C01808=1056.490,410.980,-122.148,174.990,39.875,157.709
C01809=1056.498,411.227,-122.192,174.998,39.884,157.712
C01810=1056.506,411.473,-122.237,175.006,39.892,157.714
C01811=1056.516,411.718,-122.281,175.013,39.901,157.717
C01812=1056.525,411.964,-122.327,175.022,39.910,157.719
C01813=1056.534,412.210,-122.372,175.029,39.918,157.722
C01814=1056.543,412.455,-122.416,175.037,39.927,157.724
C01815=1056.552,412.702,-122.461,175.045,39.935,157.727
C01816=1056.561,412.947,-122.506,175.053,39.944,157.730
C01817=1056.570,413.193,-122.552,175.062,39.953,157.732
C01818=1056.579,413.439,-122.596,175.069,39.962,157.735
C01819=1056.588,413.685,-122.641,175.077,39.970,157.737
C01820=1056.596,413.930,-122.686,175.086,39.980,157.740
C01821=1056.605,414.176,-122.732,175.093,39.989,157.743
C01822=1056.614,414.422,-122.777,175.102,39.997,157.745
C01823=1056.623,414.668,-122.822,175.110,40.007,157.748
C01824=1056.632,414.914,-122.868,175.118,40.015,157.750
C01825=1056.641,415.159,-122.913,175.126,40.025,157.753
C01826=1056.650,415.405,-122.959,175.135,40.033,157.756
C01827=1056.659,415.650,-123.004,175.143,40.043,157.758
C01828=1056.668,415.896,-123.050,175.151,40.052,157.761
C01829=1056.680,416.243,-123.114,175.163,40.065,157.765
C01830=1056.694,416.590,-123.179,175.174,40.078,157.769
C01831=1056.706,416.937,-123.244,175.186,40.090,157.772
C01832=1056.719,417.283,-123.308,175.198,40.103,157.776
C01833=1056.728,417.529,-123.354,175.207,40.112,157.779
C01834=1056.737,417.774,-123.400,175.216,40.122,157.782
C01835=1056.746,418.020,-123.445,175.224,40.131,157.785
C01836=1056.756,418.265,-123.491,175.233,40.141,157.787
C01837=1056.765,418.512,-123.537,175.241,40.150,157.790
C01838=1056.774,418.757,-123.583,175.249,40.159,157.793
C01839=1056.783,419.002,-123.630,175.258,40.169,157.796
C01840=1056.792,419.248,-123.675,175.267,40.178,157.798
C01841=1056.801,419.493,-123.722,175.276,40.188,157.801
C01842=1056.811,419.739,-123.768,175.284,40.197,157.804
C01843=1056.820,419.985,-123.814,175.293,40.207,157.807
C01844=1056.830,420.230,-123.860,175.302,40.216,157.810
C01845=1056.839,420.476,-123.907,175.311,40.225,157.813
C01846=1056.848,420.721,-123.954,175.319,40.235,157.815
C01847=1056.857,420.967,-124.000,175.328,40.245,157.818
C01848=1056.866,421.212,-124.046,175.337,40.254,157.821
C01849=1056.876,421.458,-124.093,175.346,40.264,157.824
C01850=1056.884,421.703,-124.140,175.355,40.274,157.827
C01851=1056.894,421.949,-124.186,175.364,40.283,157.830
C01852=1056.904,422.194,-124.233,175.373,40.293,157.833
C01853=1056.912,422.439,-124.280,175.383,40.303,157.836
C01854=1056.922,422.685,-124.326,175.392,40.313,157.839
C01855=1056.932,422.930,-124.373,175.401,40.323,157.842
C01856=1056.941,423.176,-124.420,175.409,40.333,157.845
C01857=1056.950,423.421,-124.466,175.418,40.343,157.848
C01858=1056.960,423.667,-124.514,175.427,40.353,157.851
C01859=1056.969,423.912,-124.560,175.437,40.363,157.854
C01860=1056.979,424.157,-124.607,175.447,40.372,157.857
C01861=1056.988,424.402,-124.655,175.456,40.382,157.860
C01862=1056.998,424.648,-124.701,175.465,40.393,157.863
C01863=1057.007,424.894,-124.749,175.474,40.403,157.866
C01864=1057.017,425.138,-124.796,175.484,40.413,157.869
C01865=1057.026,425.384,-124.843,175.493,40.423,157.872
C01866=1057.036,425.630,-124.890,175.502,40.433,157.875
C01867=1057.046,425.875,-124.938,175.512,40.443,157.878
C01868=1057.055,426.120,-124.985,175.521,40.453,157.882
C01869=1057.065,426.366,-125.033,175.531,40.463,157.885
C01870=1057.075,426.611,-125.080,175.541,40.474,157.888
C01871=1057.084,426.856,-125.128,175.550,40.484,157.891
C01872=1057.093,427.101,-125.175,175.560,40.495,157.894
C01873=1057.104,427.347,-125.223,175.570,40.505,157.897
C01874=1057.113,427.592,-125.270,175.579,40.515,157.901
C01875=1057.123,427.837,-125.319,175.589,40.526,157.904
C01876=1057.133,428.082,-125.366,175.598,40.537,157.907
C01877=1057.142,428.327,-125.414,175.609,40.547,157.910
C01878=1057.152,428.572,-125.462,175.618,40.558,157.914
C01879=1057.162,428.818,-125.509,175.628,40.568,157.917
C01880=1057.171,429.063,-125.558,175.638,40.579,157.920
C01881=1057.181,429.308,-125.606,175.648,40.590,157.923
C01882=1057.191,429.553,-125.654,175.659,40.600,157.927
C01883=1057.201,429.798,-125.701,175.668,40.611,157.930
C01884=1057.211,430.043,-125.750,175.678,40.622,157.933
C01885=1057.226,430.412,-125.822,175.693,40.638,157.938
C01886=1057.241,430.780,-125.896,175.709,40.654,157.943
C01887=1057.255,431.149,-125.968,175.724,40.670,157.948
C01888=1057.270,431.517,-126.041,175.739,40.687,157.954
C01889=1057.280,431.762,-126.089,175.750,40.698,157.957
C01890=1057.290,432.007,-126.138,175.760,40.709,157.960
C01891=1057.300,432.251,-126.186,175.770,40.720,157.964
C01892=1057.310,432.497,-126.235,175.781,40.731,157.967
C01893=1057.320,432.742,-126.284,175.791,40.742,157.971
C01894=1057.330,432.987,-126.332,175.802,40.753,157.974
C01895=1057.340,433.231,-126.381,175.813,40.765,157.978
C01896=1057.350,433.477,-126.430,175.822,40.776,157.981
C01897=1057.360,433.722,-126.479,175.833,40.787,157.985
C01898=1057.370,433.966,-126.528,175.844,40.798,157.988
C01899=1057.380,434.212,-126.577,175.855,40.810,157.992
C01900=1057.390,434.456,-126.626,175.865,40.821,157.996
C01901=1057.401,434.702,-126.675,175.876,40.833,157.999
C01902=1057.411,434.947,-126.724,175.887,40.843,158.003
C01903=1057.421,435.191,-126.774,175.898,40.855,158.006
C01904=1057.431,435.437,-126.823,175.909,40.867,158.010
C01905=1057.441,435.681,-126.872,175.920,40.878,158.014
C01906=1057.452,435.926,-126.921,175.931,40.890,158.017
C01907=1057.462,436.171,-126.971,175.942,40.901,158.021
C01908=1057.473,436.415,-127.020,175.952,40.913,158.025
C01909=1057.483,436.660,-127.070,175.964,40.924,158.028
C01910=1057.494,436.905,-127.119,175.975,40.936,158.032
C01911=1057.504,437.150,-127.169,175.986,40.948,158.036
C01912=1057.515,437.395,-127.218,175.998,40.959,158.040
C01913=1057.525,437.640,-127.269,176.009,40.971,158.043
C01914=1057.535,437.885,-127.318,176.021,40.983,158.047
C01915=1057.545,438.130,-127.367,176.032,40.995,158.051
C01916=1057.556,438.374,-127.418,176.043,41.007,158.055
C01917=1057.566,438.619,-127.468,176.055,41.019,158.059
C01918=1057.577,438.863,-127.518,176.066,41.031,158.063
C01919=1057.587,439.108,-127.567,176.077,41.043,158.066
C01920=1057.598,439.353,-127.618,176.089,41.055,158.070
C01921=1057.608,439.598,-127.668,176.101,41.067,158.074
C01922=1057.619,439.842,-127.718,176.112,41.079,158.078
C01923=1057.630,440.087,-127.769,176.124,41.092,158.082
C01924=1057.640,440.332,-127.820,176.135,41.104,158.086
C01925=1057.650,440.576,-127.869,176.148,41.116,158.090
C01926=1057.661,440.820,-127.919,176.159,41.128,158.094
C01927=1057.672,441.065,-127.970,176.171,41.141,158.098
C01928=1057.683,441.310,-128.020,176.183,41.153,158.102
C01929=1057.693,441.554,-128.071,176.195,41.166,158.106
C01930=1057.704,441.799,-128.122,176.208,41.178,158.110
C01931=1057.715,442.044,-128.172,176.219,41.190,158.114
C01932=1057.726,442.288,-128.224,176.232,41.203,158.118
C01933=1057.737,442.532,-128.274,176.244,41.216,158.123
C01934=1057.747,442.777,-128.325,176.257,41.228,158.127
C01935=1057.758,443.021,-128.376,176.268,41.241,158.131
C01936=1057.769,443.266,-128.428,176.281,41.254,158.135
C01937=1057.780,443.511,-128.478,176.293,41.266,158.139
C01938=1057.791,443.755,-128.529,176.306,41.279,158.143
C01939=1057.802,443.999,-128.580,176.318,41.292,158.148
C01940=1057.813,444.244,-128.632,176.330,41.305,158.152
C01941=1057.823,444.475,-128.680,176.343,41.317,158.156
C01942=1057.834,444.706,-128.729,176.355,41.329,158.160
C01943=1057.844,444.938,-128.778,176.366,41.341,158.164
C01944=1057.854,445.168,-128.826,176.378,41.354,158.168
C01945=1057.865,445.400,-128.875,176.391,41.366,158.172
C01946=1057.875,445.631,-128.924,176.403,41.378,158.176
C01947=1057.886,445.863,-128.973,176.415,41.391,158.181
C01948=1057.897,446.094,-129.022,176.427,41.404,158.185
C01949=1057.908,446.338,-129.073,176.440,41.417,158.189
C01950=1057.919,446.581,-129.125,176.453,41.430,158.193
C01951=1057.930,446.825,-129.176,176.467,41.443,158.198
C01952=1057.942,447.070,-129.228,176.480,41.456,158.202
C01953=1057.954,447.313,-129.279,176.493,41.469,158.207
C01954=1057.968,447.556,-129.329,176.506,41.482,158.211
C01955=1057.982,447.800,-129.379,176.520,41.495,158.215
C01956=1057.996,448.045,-129.428,176.533,41.507,158.220
C01957=1058.013,448.300,-129.478,176.547,41.519,158.224
C01958=1058.030,448.556,-129.529,176.562,41.532,158.228
C01959=1058.049,448.812,-129.577,176.576,41.544,158.233
C01960=1058.068,449.068,-129.626,176.590,41.556,158.237
C01961=1058.087,449.313,-129.673,176.604,41.568,158.241
C01962=1058.108,449.558,-129.718,176.618,41.578,158.245
C01963=1058.129,449.804,-129.763,176.632,41.589,158.249
C01964=1058.151,450.049,-129.807,176.646,41.600,158.252
C01965=1057.824,450.063,-130.090,176.642,41.708,158.282
C01966=1057.802,449.819,-130.046,176.628,41.698,158.279
C01967=1057.781,449.573,-130.001,176.614,41.687,158.275
C01968=1057.760,449.328,-129.956,176.600,41.676,158.271
C01969=1057.741,449.083,-129.911,176.586,41.665,158.267
C01970=1057.722,448.838,-129.864,176.572,41.653,158.263
C01971=1057.704,448.593,-129.816,176.558,41.641,158.259
C01972=1057.687,448.349,-129.769,176.545,41.630,158.255
C01973=1057.671,448.104,-129.720,176.531,41.618,158.250
C01974=1057.656,447.860,-129.672,176.517,41.606,158.246
C01975=1057.641,447.616,-129.622,176.504,41.593,158.242
C01976=1057.627,447.372,-129.572,176.491,41.581,158.238
C01977=1057.614,447.129,-129.522,176.477,41.568,158.233
C01978=1057.603,446.885,-129.470,176.464,41.555,158.229
C01979=1057.592,446.641,-129.418,176.450,41.542,158.224
C01980=1057.580,446.398,-129.367,176.437,41.528,158.220
C01981=1057.569,446.154,-129.315,176.424,41.515,158.216
C01982=1057.558,445.927,-129.267,176.412,41.503,158.211
C01983=1057.548,445.700,-129.220,176.400,41.491,158.207
C01984=1057.538,445.472,-129.171,176.388,41.479,158.203
C01985=1057.527,445.244,-129.123,176.376,41.467,158.199
C01986=1057.517,445.018,-129.076,176.364,41.455,158.195
C01987=1057.507,444.790,-129.027,176.353,41.442,158.191
C01988=1057.497,444.563,-128.980,176.340,41.430,158.187
C01989=1057.486,444.335,-128.932,176.328,41.419,158.183
C01990=1057.475,444.091,-128.880,176.315,41.406,158.179
C01991=1057.465,443.846,-128.829,176.303,41.393,158.175
C01992=1057.453,443.602,-128.778,176.291,41.380,158.171
C01993=1057.443,443.358,-128.726,176.279,41.368,158.166
C01994=1057.432,443.113,-128.676,176.266,41.355,158.162
C01995=1057.421,442.869,-128.624,176.253,41.342,158.158
C01996=1057.410,442.624,-128.574,176.241,41.330,158.154
C01997=1057.399,442.379,-128.523,176.229,41.317,158.150
C01998=1057.382,441.999,-128.444,176.210,41.298,158.143
C01999=1057.365,441.618,-128.364,176.191,41.278,158.137
C02000=1057.348,441.236,-128.286,176.172,41.259,158.131
C02001=1057.332,440.856,-128.207,176.154,41.240,158.124
C02002=1057.321,440.611,-128.156,176.141,41.228,158.120
C02003=1057.310,440.367,-128.105,176.129,41.216,158.116
C02004=1057.299,440.122,-128.055,176.118,41.203,158.112
C02005=1057.289,439.877,-128.005,176.105,41.191,158.108
C02006=1057.279,439.633,-127.955,176.094,41.179,158.104
C02007=1057.268,439.389,-127.905,176.082,41.167,158.100
C02008=1057.257,439.144,-127.855,176.071,41.155,158.096
C02009=1057.247,438.899,-127.804,176.059,41.143,158.093
C02010=1057.237,438.654,-127.754,176.047,41.131,158.089
C02011=1057.226,438.409,-127.704,176.036,41.119,158.085
C02012=1057.215,438.164,-127.655,176.024,41.107,158.081
C02013=1057.205,437.920,-127.604,176.013,41.096,158.077
C02014=1057.195,437.675,-127.554,176.002,41.084,158.074
C02015=1057.184,437.430,-127.505,175.991,41.072,158.070
C02016=1057.174,437.186,-127.456,175.979,41.060,158.066
C02017=1057.163,436.941,-127.406,175.968,41.048,158.062
C02018=1057.152,436.696,-127.356,175.957,41.037,158.058
C02019=1057.142,436.451,-127.306,175.946,41.025,158.055
C02020=1057.132,436.206,-127.257,175.934,41.014,158.051
C02021=1057.121,435.961,-127.208,175.923,41.002,158.047
C02022=1057.111,435.717,-127.159,175.912,40.991,158.044
C02023=1057.100,435.472,-127.109,175.901,40.979,158.040
C02024=1057.090,435.227,-127.060,175.890,40.967,158.036
C02025=1057.080,434.982,-127.010,175.879,40.956,158.033
C02026=1057.070,434.737,-126.962,175.868,40.945,158.029
C02027=1057.059,434.492,-126.912,175.857,40.934,158.025
C02028=1057.049,434.247,-126.863,175.847,40.922,158.022
C02029=1057.039,434.002,-126.814,175.836,40.911,158.018
C02030=1057.029,433.758,-126.765,175.825,40.900,158.015
C02031=1057.019,433.513,-126.716,175.814,40.889,158.011
C02032=1057.009,433.267,-126.667,175.804,40.877,158.008
C02033=1056.999,433.023,-126.618,175.793,40.866,158.004
C02034=1056.989,432.778,-126.569,175.782,40.855,158.001
C02035=1056.978,432.532,-126.521,175.771,40.844,157.997
C02036=1056.969,432.287,-126.472,175.762,40.833,157.994
C02037=1056.959,432.043,-126.423,175.751,40.822,157.990
C02038=1056.949,431.803,-126.375,175.741,40.811,157.987
C02039=1056.939,431.564,-126.328,175.730,40.801,157.983
C02040=1056.929,431.325,-126.280,175.720,40.790,157.980
C02041=1056.920,431.086,-126.233,175.711,40.779,157.977
C02042=1056.910,430.846,-126.186,175.700,40.769,157.973
C02043=1056.901,430.607,-126.138,175.691,40.758,157.970
C02044=1056.891,430.367,-126.092,175.680,40.748,157.967
C02045=1056.882,430.128,-126.044,175.670,40.737,157.964
C02046=1056.872,429.883,-125.996,175.661,40.726,157.960
C02047=1056.862,429.638,-125.948,175.650,40.716,157.957
C02048=1056.852,429.393,-125.900,175.640,40.705,157.954
C02049=1056.842,429.147,-125.852,175.630,40.695,157.950
C02050=1056.832,428.903,-125.804,175.620,40.684,157.947
C02051=1056.822,428.657,-125.756,175.611,40.673,157.944
C02052=1056.813,428.412,-125.708,175.600,40.663,157.940
C02053=1056.803,428.167,-125.660,175.591,40.652,157.937
C02054=1056.793,427.922,-125.612,175.580,40.642,157.934
C02055=1056.783,427.676,-125.564,175.571,40.632,157.931
C02056=1056.773,427.431,-125.517,175.561,40.621,157.928
C02057=1056.764,427.185,-125.469,175.552,40.611,157.924
C02058=1056.754,426.940,-125.421,175.541,40.601,157.921
C02059=1056.744,426.696,-125.374,175.532,40.590,157.918
C02060=1056.735,426.450,-125.326,175.522,40.580,157.915
C02061=1056.725,426.205,-125.278,175.513,40.570,157.912
C02062=1056.715,425.959,-125.231,175.503,40.559,157.908
C02063=1056.706,425.714,-125.183,175.493,40.549,157.905
C02064=1056.696,425.469,-125.136,175.484,40.539,157.902
C02065=1056.687,425.223,-125.089,175.474,40.529,157.899
C02066=1056.677,424.978,-125.042,175.465,40.519,157.896
C02067=1056.667,424.733,-124.995,175.456,40.509,157.893
C02068=1056.658,424.487,-124.947,175.447,40.499,157.890
C02069=1056.648,424.242,-124.901,175.437,40.489,157.887
C02070=1056.639,423.997,-124.853,175.428,40.479,157.884
C02071=1056.629,423.751,-124.806,175.418,40.469,157.881
C02072=1056.620,423.506,-124.760,175.408,40.459,157.878
C02073=1056.610,423.261,-124.712,175.399,40.449,157.875
C02074=1056.601,423.015,-124.666,175.390,40.439,157.872
C02075=1056.591,422.770,-124.618,175.381,40.430,157.869
C02076=1056.582,422.525,-124.572,175.372,40.420,157.866
C02077=1056.572,422.279,-124.526,175.363,40.410,157.863
C02078=1056.563,422.034,-124.478,175.354,40.400,157.860
C02079=1056.553,421.788,-124.432,175.345,40.390,157.857
C02080=1056.544,421.543,-124.386,175.336,40.381,157.854
C02081=1056.536,421.297,-124.339,175.327,40.371,157.851
C02082=1056.526,421.051,-124.292,175.318,40.361,157.848
C02083=1056.517,420.806,-124.246,175.309,40.352,157.845
C02084=1056.508,420.561,-124.199,175.300,40.342,157.842
C02085=1056.498,420.315,-124.152,175.292,40.333,157.840
C02086=1056.489,420.070,-124.105,175.283,40.323,157.837
C02087=1056.480,419.825,-124.059,175.274,40.314,157.834
C02088=1056.470,419.578,-124.014,175.265,40.304,157.831
C02089=1056.461,419.333,-123.967,175.256,40.295,157.828
C02090=1056.452,419.088,-123.921,175.248,40.285,157.825
C02091=1056.442,418.842,-123.875,175.239,40.276,157.823
C02092=1056.433,418.596,-123.829,175.230,40.267,157.820
C02093=1056.424,418.350,-123.783,175.221,40.257,157.817
C02094=1056.415,418.105,-123.737,175.213,40.248,157.814
C02095=1056.406,417.859,-123.691,175.204,40.239,157.812
C02096=1056.397,417.614,-123.645,175.195,40.230,157.809
C02097=1056.388,417.368,-123.600,175.187,40.221,157.806
C02098=1056.375,417.020,-123.534,175.175,40.207,157.802
C02099=1056.361,416.671,-123.469,175.163,40.194,157.798
C02100=1056.348,416.322,-123.405,175.151,40.182,157.794
C02101=1056.336,415.974,-123.339,175.139,40.169,157.791
C02102=1056.327,415.728,-123.294,175.130,40.160,157.788
C02103=1056.318,415.482,-123.248,175.123,40.150,157.785
C02104=1056.309,415.236,-123.203,175.114,40.142,157.783
C02105=1056.300,414.990,-123.158,175.106,40.132,157.780
C02106=1056.291,414.745,-123.112,175.097,40.124,157.777
C02107=1056.282,414.499,-123.066,175.090,40.114,157.775
C02108=1056.273,414.254,-123.021,175.081,40.106,157.772
C02109=1056.264,414.008,-122.975,175.073,40.097,157.769
C02110=1056.255,413.762,-122.930,175.065,40.088,157.767
C02111=1056.247,413.516,-122.885,175.057,40.079,157.764
C02112=1056.237,413.271,-122.841,175.048,40.070,157.762
C02113=1056.228,413.025,-122.795,175.041,40.062,157.759
C02114=1056.219,412.779,-122.750,175.033,40.053,157.757
C02115=1056.211,412.533,-122.705,175.024,40.044,157.754
C02116=1056.201,412.287,-122.660,175.017,40.036,157.751
C02117=1056.192,412.041,-122.615,175.008,40.027,157.749
C02118=1056.184,411.795,-122.570,175.001,40.019,157.746
C02119=1056.174,411.550,-122.526,174.993,40.010,157.744
C02120=1056.165,411.304,-122.480,174.984,40.001,157.741
C02121=1056.157,411.058,-122.436,174.977,39.993,157.739
C02122=1056.148,410.813,-122.390,174.969,39.984,157.736
C02123=1056.139,410.566,-122.346,174.961,39.976,157.734
C02124=1056.131,410.321,-122.302,174.953,39.967,157.731
C02125=1056.122,410.075,-122.257,174.946,39.959,157.729
C02126=1056.112,409.829,-122.213,174.938,39.950,157.727
C02127=1056.104,409.583,-122.168,174.930,39.942,157.724
C02128=1056.095,409.337,-122.123,174.922,39.933,157.722
C02129=1056.086,409.092,-122.079,174.915,39.925,157.719
C02130=1056.078,408.845,-122.034,174.907,39.917,157.717
C02131=1056.069,408.600,-121.991,174.899,39.908,157.714
C02132=1056.060,408.353,-121.946,174.891,39.900,157.712
C02133=1056.052,408.108,-121.902,174.884,39.892,157.710
C02134=1056.043,407.862,-121.857,174.876,39.883,157.707
C02135=1056.034,407.616,-121.812,174.869,39.875,157.705
C02136=1056.026,407.370,-121.768,174.862,39.867,157.702
C02137=1056.017,407.124,-121.724,174.853,39.859,157.700
C02138=1056.009,406.878,-121.680,174.846,39.850,157.698
C02139=1056.000,406.632,-121.636,174.839,39.842,157.695
C02140=1055.992,406.386,-121.592,174.831,39.834,157.693
C02141=1055.984,406.140,-121.548,174.824,39.826,157.691
C02142=1055.974,405.894,-121.503,174.816,39.818,157.688
C02143=1055.966,405.649,-121.459,174.809,39.810,157.686
C02144=1055.958,405.403,-121.416,174.802,39.801,157.684
C02145=1055.950,405.157,-121.372,174.794,39.793,157.681
C02146=1055.940,404.911,-121.328,174.787,39.786,157.679
C02147=1055.932,404.664,-121.284,174.780,39.777,157.677
C02148=1055.924,404.419,-121.240,174.773,39.769,157.674
C02149=1055.916,404.173,-121.196,174.765,39.762,157.672
C02150=1055.906,403.926,-121.152,174.758,39.754,157.670
C02151=1055.898,403.680,-121.109,174.751,39.745,157.668
C02152=1055.890,403.435,-121.065,174.743,39.738,157.665
C02153=1055.881,403.189,-121.022,174.736,39.730,157.663
C02154=1055.870,402.846,-120.961,174.726,39.719,157.660
C02155=1055.857,402.503,-120.901,174.716,39.708,157.657
C02156=1055.846,402.160,-120.840,174.706,39.697,157.654
C02157=1055.835,401.817,-120.780,174.697,39.686,157.651
C02158=1055.826,401.570,-120.736,174.690,39.679,157.649
C02159=1055.817,401.325,-120.693,174.683,39.671,157.646
C02160=1055.809,401.079,-120.650,174.675,39.663,157.644
C02161=1055.800,400.833,-120.606,174.668,39.656,157.642
C02162=1055.792,400.586,-120.563,174.661,39.648,157.640
C02163=1055.784,400.340,-120.520,174.654,39.640,157.638
C02164=1055.775,400.094,-120.477,174.647,39.633,157.636
C02165=1055.767,399.848,-120.434,174.641,39.626,157.634
C02166=1055.758,399.602,-120.391,174.634,39.618,157.631
C02167=1055.750,399.356,-120.348,174.627,39.611,157.629
C02168=1055.742,399.110,-120.306,174.620,39.603,157.627
C02169=1055.734,398.864,-120.262,174.612,39.595,157.625
C02170=1055.726,398.618,-120.219,174.606,39.588,157.623
C02171=1055.717,398.371,-120.176,174.599,39.581,157.621
C02172=1055.709,398.125,-120.133,174.592,39.573,157.619
C02173=1055.701,397.879,-120.091,174.585,39.565,157.617
C02174=1055.693,397.633,-120.048,174.579,39.558,157.615
C02175=1055.684,397.387,-120.005,174.572,39.551,157.612
C02176=1055.676,397.141,-119.963,174.565,39.543,157.610
C02177=1055.668,396.895,-119.920,174.558,39.536,157.608
C02178=1055.660,396.649,-119.878,174.552,39.529,157.606
C02179=1055.652,396.403,-119.835,174.545,39.521,157.604
C02180=1055.643,396.156,-119.792,174.538,39.514,157.602
C02181=1055.635,395.910,-119.749,174.532,39.507,157.600
C02182=1055.627,395.664,-119.707,174.525,39.500,157.598
C02183=1055.619,395.418,-119.664,174.518,39.492,157.596
C02184=1055.611,395.171,-119.622,174.512,39.485,157.594
C02185=1055.603,394.925,-119.580,174.505,39.478,157.592
C02186=1055.594,394.679,-119.538,174.498,39.471,157.590
C02187=1055.586,394.433,-119.495,174.493,39.464,157.588
C02188=1055.578,394.187,-119.454,174.486,39.456,157.586
C02189=1055.570,393.940,-119.411,174.479,39.450,157.584
C02190=1055.562,393.695,-119.369,174.473,39.442,157.582
C02191=1055.554,393.448,-119.326,174.466,39.435,157.580
C02192=1055.546,393.202,-119.284,174.460,39.428,157.578
C02193=1055.537,392.956,-119.243,174.453,39.421,157.576
C02194=1055.530,392.710,-119.201,174.446,39.414,157.574
C02195=1055.521,392.463,-119.158,174.440,39.407,157.572
C02196=1055.514,392.217,-119.116,174.433,39.400,157.570
C02197=1055.505,391.971,-119.075,174.428,39.393,157.569
C02198=1055.497,391.725,-119.033,174.421,39.386,157.567
C02199=1055.489,391.478,-118.990,174.415,39.379,157.565
C02200=1055.481,391.232,-118.948,174.408,39.372,157.563
C02201=1055.472,390.986,-118.907,174.401,39.366,157.561
C02202=1055.465,390.739,-118.866,174.395,39.359,157.559
C02203=1055.458,390.493,-118.824,174.389,39.352,157.557
C02204=1055.449,390.247,-118.782,174.383,39.345,157.555
C02205=1055.441,390.001,-118.740,174.376,39.338,157.553
C02206=1055.433,389.754,-118.698,174.370,39.331,157.551
C02207=1055.425,389.508,-118.657,174.363,39.324,157.550
C02208=1055.417,389.262,-118.615,174.358,39.318,157.548
C02209=1055.409,389.015,-118.574,174.352,39.311,157.546
C02210=1055.398,388.689,-118.519,174.344,39.302,157.543
C02211=1055.388,388.365,-118.465,174.335,39.293,157.541
C02212=1055.377,388.040,-118.410,174.327,39.284,157.539
C02213=1055.366,387.714,-118.356,174.319,39.275,157.536
C02214=1055.359,387.468,-118.314,174.313,39.269,157.534
C02215=1055.350,387.221,-118.273,174.306,39.262,157.533
C02216=1055.343,386.975,-118.232,174.301,39.256,157.531
C02217=1055.334,386.729,-118.190,174.294,39.249,157.529
C02218=1055.327,386.483,-118.149,174.288,39.242,157.527
C02219=1055.319,386.236,-118.109,174.282,39.236,157.525
C02220=1055.310,385.989,-118.068,174.276,39.230,157.524
C02221=1055.303,385.743,-118.026,174.270,39.223,157.522
C02222=1055.295,385.497,-117.985,174.263,39.216,157.520
C02223=1055.288,385.251,-117.944,174.258,39.210,157.518
C02224=1055.279,385.004,-117.903,174.252,39.204,157.517
C02225=1055.271,384.758,-117.862,174.245,39.197,157.515
C02226=1055.264,384.511,-117.821,174.240,39.190,157.513
C02227=1055.256,384.264,-117.780,174.234,39.184,157.511
C02228=1055.248,384.018,-117.740,174.227,39.177,157.509
C02229=1055.240,383.771,-117.698,174.222,39.171,157.508
C02230=1055.232,383.525,-117.658,174.216,39.165,157.506
C02231=1055.225,383.279,-117.617,174.211,39.158,157.504
C02232=1055.217,383.032,-117.576,174.204,39.152,157.502
C02233=1055.209,382.786,-117.535,174.198,39.145,157.501
C02234=1055.202,382.539,-117.494,174.193,39.139,157.499
C02235=1055.194,382.293,-117.454,174.187,39.133,157.497
C02236=1055.186,382.046,-117.413,174.181,39.126,157.496
C02237=1055.179,381.800,-117.372,174.175,39.120,157.494
C02238=1055.171,381.553,-117.332,174.169,39.114,157.492
C02239=1055.163,381.307,-117.291,174.164,39.107,157.491
C02240=1055.156,381.061,-117.251,174.157,39.101,157.489
C02241=1055.148,380.814,-117.210,174.152,39.095,157.487
C02242=1055.140,380.568,-117.170,174.146,39.089,157.485
C02243=1055.133,380.321,-117.129,174.141,39.082,157.484
C02244=1055.125,380.075,-117.088,174.135,39.076,157.482
C02245=1055.117,379.828,-117.048,174.128,39.070,157.480
C02246=1055.109,379.581,-117.008,174.123,39.064,157.479
C02247=1055.102,379.334,-116.968,174.117,39.058,157.477
C02248=1055.094,379.088,-116.928,174.112,39.052,157.476
C02249=1055.086,378.841,-116.887,174.106,39.045,157.474
C02250=1055.079,378.595,-116.848,174.100,39.039,157.472
C02251=1055.071,378.349,-116.807,174.094,39.034,157.471
C02252=1055.063,378.102,-116.767,174.089,39.027,157.469
C02253=1055.055,377.855,-116.727,174.083,39.021,157.467
C02254=1055.048,377.608,-116.687,174.078,39.015,157.466
C02255=1055.040,377.362,-116.647,174.072,39.009,157.464
C02256=1055.032,377.116,-116.607,174.067,39.003,157.462
C02257=1055.025,376.869,-116.567,174.060,38.997,157.461
C02258=1055.017,376.622,-116.527,174.055,38.991,157.459
C02259=1055.009,376.375,-116.487,174.050,38.985,157.458
C02260=1055.002,376.129,-116.448,174.044,38.979,157.456
C02261=1054.994,375.882,-116.407,174.039,38.973,157.455
C02262=1054.986,375.635,-116.367,174.033,38.968,157.453
C02263=1054.979,375.389,-116.328,174.028,38.962,157.451
C02264=1054.972,375.142,-116.288,174.022,38.956,157.450
C02265=1054.964,374.895,-116.248,174.017,38.950,157.448
C02266=1054.955,374.602,-116.201,174.010,38.942,157.446
C02267=1054.946,374.309,-116.154,174.003,38.935,157.444
C02268=1054.937,374.016,-116.107,173.997,38.928,157.443
C02269=1054.929,373.722,-116.060,173.991,38.922,157.441
C02270=1054.921,373.475,-116.020,173.986,38.916,157.439
C02271=1054.913,373.228,-115.980,173.980,38.910,157.438
C02272=1054.906,372.982,-115.941,173.975,38.904,157.436
C02273=1054.898,372.735,-115.901,173.969,38.898,157.435
C02274=1054.891,372.488,-115.862,173.964,38.892,157.433
C02275=1054.884,372.242,-115.822,173.959,38.887,157.432
C02276=1054.877,371.995,-115.783,173.953,38.881,157.430
C02277=1054.869,371.748,-115.743,173.948,38.875,157.428
C02278=1054.861,371.502,-115.704,173.943,38.869,157.427
C02279=1054.854,371.255,-115.665,173.937,38.863,157.425
C02280=1054.846,371.008,-115.625,173.932,38.858,157.424
C02281=1054.838,370.762,-115.586,173.927,38.852,157.422
C02282=1054.831,370.514,-115.547,173.921,38.847,157.421
C02283=1054.823,370.268,-115.508,173.916,38.841,157.419
C02284=1054.816,370.021,-115.469,173.911,38.835,157.418
C02285=1054.809,369.774,-115.429,173.905,38.830,157.417
C02286=1054.800,369.527,-115.391,173.900,38.824,157.415
C02287=1054.794,369.280,-115.352,173.895,38.819,157.414
C02288=1054.786,369.034,-115.312,173.889,38.813,157.412
C02289=1054.778,368.787,-115.274,173.884,38.807,157.411
C02290=1054.771,368.540,-115.235,173.879,38.802,157.409
C02291=1054.763,368.294,-115.196,173.873,38.797,157.408
C02292=1054.756,368.047,-115.157,173.868,38.791,157.406
C02293=1054.749,367.800,-115.118,173.864,38.785,157.405
C02294=1054.741,367.553,-115.079,173.858,38.780,157.403
C02295=1054.734,367.307,-115.040,173.853,38.774,157.402
C02296=1054.727,367.060,-115.002,173.848,38.769,157.401
C02297=1054.719,366.812,-114.962,173.843,38.763,157.399
C02298=1054.712,366.566,-114.924,173.837,38.757,157.398
C02299=1054.705,366.319,-114.885,173.832,38.752,157.396
C02300=1054.697,366.072,-114.846,173.827,38.747,157.395
C02301=1054.690,365.825,-114.808,173.822,38.741,157.393
C02302=1054.683,365.578,-114.769,173.817,38.736,157.392
C02303=1054.675,365.331,-114.730,173.812,38.730,157.390
C02304=1054.668,365.084,-114.692,173.807,38.725,157.389
C02305=1054.661,364.837,-114.653,173.801,38.719,157.388
C02306=1054.654,364.591,-114.615,173.797,38.714,157.386
C02307=1054.647,364.344,-114.576,173.792,38.709,157.385
C02308=1054.639,364.097,-114.537,173.787,38.703,157.383
C02309=1054.632,363.850,-114.498,173.781,38.698,157.382
C02310=1054.624,363.604,-114.460,173.776,38.692,157.381
C02311=1054.618,363.356,-114.422,173.772,38.687,157.379
C02312=1054.610,363.110,-114.384,173.767,38.682,157.378
C02313=1054.602,362.862,-114.345,173.762,38.677,157.377
C02314=1054.595,362.616,-114.306,173.756,38.671,157.375
C02315=1054.588,362.368,-114.269,173.751,38.666,157.374
C02316=1054.581,362.122,-114.230,173.747,38.661,157.372
C02317=1054.574,361.875,-114.192,173.742,38.655,157.371
C02318=1054.567,361.628,-114.154,173.737,38.650,157.370
C02319=1054.558,361.381,-114.115,173.731,38.645,157.368
C02320=1054.552,361.133,-114.077,173.727,38.640,157.367
C02321=1054.544,360.887,-114.039,173.722,38.635,157.366
C02322=1054.536,360.612,-113.997,173.717,38.629,157.364
C02323=1054.528,360.337,-113.954,173.712,38.623,157.363
C02324=1054.521,360.063,-113.912,173.706,38.617,157.361
C02325=1054.512,359.788,-113.871,173.700,38.612,157.360
C02326=1054.505,359.541,-113.832,173.696,38.606,157.358
C02327=1054.498,359.294,-113.794,173.691,38.601,157.357
C02328=1054.490,359.048,-113.756,173.685,38.596,157.356
C02329=1054.483,358.801,-113.719,173.681,38.591,157.354
C02330=1054.477,358.553,-113.681,173.676,38.586,157.353
C02331=1054.469,358.307,-113.642,173.671,38.581,157.352
C02332=1054.462,358.059,-113.605,173.667,38.576,157.350
C02333=1054.455,357.812,-113.567,173.662,38.570,157.349
C02334=1054.447,357.565,-113.530,173.657,38.565,157.348
C02335=1054.440,357.319,-113.492,173.652,38.560,157.347
C02336=1054.432,357.072,-113.454,173.647,38.555,157.345
C02337=1054.425,356.824,-113.416,173.642,38.551,157.344
C02338=1054.418,356.577,-113.379,173.638,38.545,157.343
C02339=1054.411,356.330,-113.341,173.633,38.540,157.341
C02340=1054.404,356.083,-113.304,173.628,38.535,157.340
C02341=1054.397,355.836,-113.266,173.624,38.530,157.339
C02342=1054.390,355.588,-113.228,173.619,38.525,157.338
C02343=1054.383,355.341,-113.191,173.615,38.520,157.336
C02344=1054.375,355.094,-113.153,173.610,38.516,157.335
C02345=1054.368,354.847,-113.116,173.604,38.511,157.334
C02346=1054.361,354.600,-113.078,173.600,38.506,157.333
C02347=1054.354,354.353,-113.041,173.595,38.500,157.331
C02348=1054.347,354.106,-113.003,173.591,38.495,157.330
C02349=1054.340,353.859,-112.966,173.586,38.490,157.329
C02350=1054.332,353.612,-112.928,173.581,38.485,157.327
C02351=1054.325,353.365,-112.891,173.577,38.480,157.326
C02352=1054.318,353.117,-112.854,173.572,38.476,157.325
C02353=1054.312,352.871,-112.817,173.568,38.471,157.324
C02354=1054.304,352.624,-112.779,173.563,38.466,157.322
C02355=1054.297,352.376,-112.742,173.559,38.461,157.321
C02356=1054.289,352.129,-112.706,173.554,38.456,157.320
C02357=1054.282,351.882,-112.668,173.549,38.451,157.319
C02358=1054.276,351.635,-112.631,173.544,38.446,157.317
C02359=1054.268,351.388,-112.593,173.539,38.442,157.316
C02360=1054.261,351.141,-112.557,173.535,38.437,157.315
C02361=1054.255,350.894,-112.519,173.530,38.432,157.314
C02362=1054.248,350.646,-112.483,173.526,38.427,157.313
C02363=1054.241,350.399,-112.445,173.521,38.422,157.311
C02364=1054.233,350.152,-112.409,173.517,38.418,157.310
C02365=1054.226,349.905,-112.372,173.512,38.413,157.309
C02366=1054.219,349.658,-112.335,173.508,38.408,157.308
C02367=1054.212,349.410,-112.297,173.503,38.404,157.307
C02368=1054.204,349.163,-112.261,173.499,38.399,157.305
C02369=1054.198,348.917,-112.224,173.494,38.394,157.304
C02370=1054.191,348.669,-112.187,173.490,38.389,157.303
C02371=1054.183,348.422,-112.150,173.485,38.384,157.302
C02372=1054.176,348.175,-112.114,173.481,38.380,157.301
C02373=1054.170,347.927,-112.077,173.476,38.375,157.299
C02374=1054.163,347.681,-112.040,173.472,38.371,157.298
C02375=1054.155,347.433,-112.004,173.467,38.366,157.297
C02376=1054.148,347.186,-111.967,173.463,38.361,157.296
C02377=1054.142,346.939,-111.930,173.459,38.356,157.295
C02378=1054.134,346.669,-111.890,173.454,38.351,157.293
C02379=1054.126,346.399,-111.850,173.449,38.346,157.292
C02380=1054.118,346.130,-111.810,173.444,38.341,157.291
C02381=1054.111,345.860,-111.770,173.440,38.336,157.290
C02382=1054.104,345.613,-111.735,173.435,38.331,157.288
C02383=1054.097,345.366,-111.697,173.431,38.326,157.287
C02384=1054.090,345.119,-111.661,173.426,38.322,157.286
C02385=1054.083,344.871,-111.624,173.422,38.318,157.285
C02386=1054.076,344.624,-111.588,173.418,38.313,157.284
C02387=1054.069,344.377,-111.552,173.413,38.308,157.283
C02388=1054.062,344.130,-111.515,173.409,38.304,157.281
C02389=1054.055,343.882,-111.478,173.404,38.299,157.280
C02390=1054.048,343.635,-111.443,173.400,38.294,157.279
C02391=1054.041,343.387,-111.406,173.396,38.290,157.278
C02392=1054.034,343.141,-111.370,173.391,38.286,157.277
C02393=1054.027,342.893,-111.333,173.387,38.281,157.276
C02394=1054.020,342.646,-111.297,173.383,38.276,157.275
C02395=1054.013,342.398,-111.260,173.378,38.272,157.273
C02396=1054.007,342.151,-111.225,173.374,38.267,157.272
C02397=1053.999,341.904,-111.189,173.370,38.263,157.271
C02398=1053.993,341.657,-111.153,173.366,38.258,157.270
C02399=1053.985,341.409,-111.116,173.362,38.254,157.269
C02400=1053.979,341.162,-111.081,173.357,38.250,157.268
C02401=1053.972,340.915,-111.045,173.353,38.245,157.267
C02402=1053.964,340.667,-111.009,173.349,38.240,157.266
C02403=1053.958,340.420,-110.972,173.344,38.236,157.265
C02404=1053.950,340.172,-110.937,173.340,38.231,157.263
C02405=1053.943,339.925,-110.901,173.336,38.227,157.262
C02406=1053.937,339.678,-110.864,173.331,38.222,157.261
C02407=1053.930,339.430,-110.829,173.327,38.218,157.260
C02408=1053.923,339.184,-110.793,173.323,38.213,157.259
C02409=1053.917,338.936,-110.757,173.319,38.209,157.258
C02410=1053.909,338.688,-110.721,173.315,38.205,157.257
C02411=1053.902,338.441,-110.686,173.311,38.200,157.256
C02412=1053.896,338.194,-110.650,173.307,38.196,157.255
C02413=1053.888,337.947,-110.613,173.302,38.192,157.254
C02414=1053.881,337.699,-110.578,173.298,38.187,157.253
C02415=1053.875,337.452,-110.542,173.294,38.183,157.251
C02416=1053.868,337.205,-110.507,173.290,38.179,157.250
C02417=1053.861,336.957,-110.471,173.285,38.174,157.249
C02418=1053.855,336.710,-110.435,173.281,38.170,157.248
C02419=1053.848,336.462,-110.400,173.278,38.165,157.247
C02420=1053.841,336.216,-110.364,173.274,38.161,157.246
C02421=1053.833,335.968,-110.328,173.269,38.157,157.245
C02422=1053.827,335.720,-110.293,173.265,38.152,157.244
C02423=1053.820,335.473,-110.258,173.261,38.148,157.243
C02424=1053.813,335.226,-110.222,173.257,38.144,157.242
C02425=1053.806,334.978,-110.186,173.252,38.140,157.241
C02426=1053.799,334.730,-110.151,173.249,38.135,157.240
C02427=1053.793,334.483,-110.116,173.245,38.131,157.239
C02428=1053.786,334.236,-110.080,173.241,38.127,157.238
C02429=1053.779,333.989,-110.045,173.236,38.122,157.236
C02430=1053.771,333.741,-110.009,173.232,38.118,157.236
C02431=1053.765,333.493,-109.974,173.228,38.114,157.234
C02432=1053.758,333.246,-109.939,173.224,38.110,157.233
C02433=1053.751,332.999,-109.904,173.221,38.106,157.232
C02434=1053.743,332.725,-109.864,173.216,38.101,157.231
C02435=1053.736,332.452,-109.826,173.212,38.096,157.230
C02436=1053.728,332.178,-109.786,173.207,38.092,157.229
C02437=1053.720,331.904,-109.748,173.203,38.087,157.228
C02438=1053.714,331.656,-109.712,173.198,38.083,157.227
C02439=1053.708,331.409,-109.677,173.194,38.078,157.226
C02440=1053.701,331.161,-109.642,173.190,38.074,157.225
C02441=1053.694,330.914,-109.606,173.187,38.070,157.224
C02442=1053.687,330.667,-109.571,173.183,38.065,157.223
C02443=1053.681,330.419,-109.536,173.179,38.062,157.222
C02444=1053.674,330.172,-109.501,173.175,38.057,157.220
C02445=1053.667,329.924,-109.467,173.170,38.053,157.220
C02446=1053.660,329.677,-109.432,173.166,38.049,157.219
C02447=1053.653,329.429,-109.397,173.163,38.045,157.217
C02448=1053.646,329.182,-109.362,173.159,38.041,157.217
C02449=1053.639,328.934,-109.328,173.155,38.037,157.216
C02450=1053.632,328.687,-109.293,173.151,38.032,157.214
C02451=1053.626,328.440,-109.258,173.147,38.029,157.214
C02452=1053.617,328.192,-109.223,173.143,38.025,157.213
C02453=1053.611,327.944,-109.188,173.139,38.021,157.212
C02454=1053.604,327.696,-109.153,173.135,38.016,157.211
C02455=1053.597,327.449,-109.119,173.131,38.012,157.210
C02456=1053.590,327.201,-109.084,173.127,38.008,157.209
C02457=1053.583,326.954,-109.049,173.124,38.005,157.208
C02458=1053.576,326.706,-109.015,173.120,38.001,157.207
C02459=1053.570,326.459,-108.980,173.116,37.996,157.206
C02460=1053.562,326.211,-108.946,173.111,37.992,157.205
C02461=1053.556,325.964,-108.911,173.108,37.988,157.204
C02462=1053.550,325.717,-108.877,173.104,37.984,157.203
C02463=1053.542,325.470,-108.843,173.100,37.980,157.202
C02464=1053.536,325.222,-108.808,173.096,37.977,157.201
C02465=1053.529,324.974,-108.773,173.092,37.972,157.200
C02466=1053.522,324.727,-108.739,173.089,37.968,157.199
C02467=1053.515,324.479,-108.704,173.085,37.964,157.198
C02468=1053.508,324.232,-108.670,173.081,37.960,157.197
C02469=1053.501,323.984,-108.636,173.077,37.956,157.196
C02470=1053.495,323.736,-108.601,173.074,37.952,157.195
C02471=1053.487,323.489,-108.567,173.070,37.948,157.194
C02472=1053.481,323.242,-108.532,173.066,37.945,157.193
C02473=1053.474,322.994,-108.498,173.062,37.940,157.192
C02474=1053.464,322.612,-108.445,173.056,37.934,157.191
C02475=1053.453,322.228,-108.392,173.050,37.928,157.189
C02476=1053.443,321.845,-108.338,173.045,37.922,157.188
C02477=1053.432,321.462,-108.287,173.039,37.916,157.186
C02478=1053.426,321.215,-108.251,173.035,37.912,157.185
C02479=1053.419,320.968,-108.218,173.031,37.908,157.184
C02480=1053.413,320.720,-108.184,173.027,37.904,157.183
C02481=1053.406,320.472,-108.149,173.024,37.900,157.182
C02482=1053.399,320.224,-108.115,173.020,37.896,157.182
C02483=1053.393,319.977,-108.081,173.016,37.892,157.181
C02484=1053.386,319.730,-108.047,173.012,37.888,157.180
C02485=1053.379,319.482,-108.012,173.009,37.884,157.179
C02486=1053.369,319.091,-107.959,173.003,37.878,157.177
C02487=1053.358,318.699,-107.905,172.997,37.872,157.176
C02488=1053.348,318.308,-107.852,172.991,37.866,157.174
C02489=1053.337,317.916,-107.798,172.985,37.860,157.173
C02490=1053.331,317.669,-107.764,172.982,37.856,157.172
C02491=1053.324,317.421,-107.730,172.979,37.852,157.171
C02492=1053.318,317.174,-107.696,172.975,37.848,157.170
C02493=1053.311,316.926,-107.662,172.971,37.844,157.169
C02494=1053.305,316.679,-107.628,172.967,37.840,157.168
C02495=1053.298,316.432,-107.594,172.964,37.836,157.167
C02496=1053.292,316.184,-107.560,172.960,37.832,157.166
C02497=1053.285,315.937,-107.526,172.956,37.828,157.165
C02498=1053.279,315.689,-107.492,172.952,37.824,157.164
C02499=1053.272,315.441,-107.459,172.949,37.821,157.163
C02500=1053.266,315.193,-107.425,172.945,37.817,157.162
C02501=1053.259,314.946,-107.391,172.942,37.813,157.162
C02502=1053.253,314.698,-107.357,172.939,37.809,157.161
C02503=1053.246,314.451,-107.323,172.935,37.805,157.160
C02504=1053.239,314.203,-107.290,172.931,37.801,157.159
C02505=1053.233,313.956,-107.256,172.927,37.797,157.158
C02506=1053.226,313.708,-107.222,172.924,37.793,157.157
C02507=1053.220,313.461,-107.188,172.920,37.790,157.156
C02508=1053.213,313.212,-107.155,172.917,37.786,157.155
C02509=1053.207,312.965,-107.122,172.914,37.782,157.154
C02510=1053.200,312.717,-107.089,172.910,37.778,157.153
C02511=1053.193,312.469,-107.055,172.906,37.774,157.152
C02512=1053.186,312.222,-107.022,172.903,37.771,157.152
C02513=1053.179,311.974,-106.988,172.899,37.767,157.151
C02514=1053.173,311.726,-106.955,172.895,37.763,157.150
C02515=1053.166,311.479,-106.922,172.892,37.760,157.149
C02516=1053.159,311.231,-106.889,172.888,37.756,157.148
C02517=1053.152,310.984,-106.855,172.885,37.752,157.147
C02518=1053.146,310.736,-106.822,172.882,37.749,157.146
C02519=1053.139,310.488,-106.789,172.878,37.745,157.145
C02520=1053.132,310.241,-106.756,172.874,37.741,157.145
C02521=1053.126,309.992,-106.723,172.871,37.737,157.144
C02522=1053.119,309.745,-106.689,172.867,37.733,157.143
C02523=1053.111,309.497,-106.657,172.863,37.730,157.142
C02524=1053.105,309.250,-106.624,172.861,37.727,157.141
C02525=1053.098,309.003,-106.590,172.857,37.723,157.140
C02526=1053.092,308.755,-106.557,172.853,37.719,157.139
C02527=1053.085,308.507,-106.525,172.850,37.715,157.138
C02528=1053.078,308.259,-106.491,172.846,37.712,157.138
C02529=1053.072,308.012,-106.458,172.842,37.708,157.137
C02530=1053.065,307.764,-106.425,172.840,37.704,157.136
C02531=1053.059,307.516,-106.392,172.836,37.701,157.135
C02532=1053.052,307.268,-106.359,172.832,37.697,157.134
C02533=1053.044,307.021,-106.326,172.829,37.693,157.133
C02534=1053.038,306.773,-106.294,172.825,37.690,157.132
C02535=1053.032,306.526,-106.261,172.822,37.686,157.132
C02536=1053.025,306.277,-106.228,172.819,37.682,157.131
C02537=1053.019,306.030,-106.195,172.815,37.679,157.130
C02538=1053.012,305.782,-106.162,172.811,37.675,157.129
C02539=1053.005,305.535,-106.128,172.808,37.672,157.128
C02540=1052.999,305.287,-106.096,172.805,37.668,157.127
C02541=1052.992,305.040,-106.063,172.802,37.664,157.126
C02542=1052.985,304.765,-106.027,172.798,37.660,157.126
C02543=1052.977,304.489,-105.991,172.794,37.656,157.125
C02544=1052.970,304.215,-105.955,172.790,37.652,157.124
C02545=1052.963,303.940,-105.918,172.787,37.648,157.123
C02546=1052.956,303.693,-105.886,172.783,37.644,157.122
C02547=1052.950,303.445,-105.853,172.779,37.641,157.121
C02548=1052.943,303.197,-105.820,172.776,37.637,157.120
C02549=1052.937,302.949,-105.787,172.773,37.633,157.119
C02550=1052.931,302.702,-105.754,172.769,37.630,157.118
C02551=1052.924,302.454,-105.722,172.766,37.626,157.118
C02552=1052.917,302.207,-105.689,172.763,37.623,157.117
C02553=1052.910,301.959,-105.656,172.759,37.619,157.116
C02554=1052.904,301.711,-105.623,172.756,37.615,157.115
C02555=1052.898,301.463,-105.591,172.752,37.612,157.114
C02556=1052.892,301.215,-105.559,172.750,37.608,157.113
C02557=1052.885,300.968,-105.527,172.746,37.604,157.112
C02558=1052.879,300.720,-105.494,172.742,37.601,157.112
C02559=1052.872,300.472,-105.461,172.740,37.597,157.111
C02560=1052.865,300.224,-105.428,172.736,37.593,157.110
C02561=1052.859,299.976,-105.396,172.733,37.590,157.109
C02562=1052.852,299.729,-105.364,172.730,37.586,157.108
C02563=1052.846,299.481,-105.331,172.726,37.583,157.107
C02564=1052.840,299.234,-105.298,172.723,37.579,157.107
C02565=1052.834,298.985,-105.266,172.720,37.575,157.106
C02566=1052.828,298.738,-105.234,172.716,37.572,157.105
C02567=1052.820,298.491,-105.201,172.713,37.568,157.104
C02568=1052.814,298.242,-105.169,172.710,37.564,157.103
C02569=1052.808,297.995,-105.137,172.706,37.561,157.102
C02570=1052.802,297.747,-105.104,172.703,37.557,157.102
C02571=1052.795,297.499,-105.072,172.700,37.554,157.101
C02572=1052.789,297.252,-105.040,172.697,37.550,157.100
C02573=1052.783,297.004,-105.008,172.693,37.547,157.099
C02574=1052.777,296.756,-104.975,172.690,37.543,157.098
C02575=1052.770,296.508,-104.942,172.687,37.539,157.097
C02576=1052.764,296.260,-104.911,172.684,37.536,157.097
C02577=1052.757,296.012,-104.878,172.681,37.532,157.096
C02578=1052.750,295.764,-104.846,172.677,37.529,157.095
C02579=1052.744,295.516,-104.814,172.674,37.525,157.094
C02580=1052.737,295.269,-104.782,172.671,37.522,157.093
C02581=1052.731,295.021,-104.750,172.667,37.518,157.092
C02582=1052.724,294.773,-104.718,172.665,37.514,157.092
C02583=1052.718,294.525,-104.686,172.661,37.511,157.091
C02584=1052.711,294.277,-104.654,172.658,37.508,157.090
C02585=1052.704,294.030,-104.622,172.655,37.504,157.089
C02586=1052.698,293.782,-104.590,172.651,37.501,157.089
C02587=1052.691,293.534,-104.559,172.649,37.497,157.088
C02588=1052.685,293.286,-104.526,172.645,37.494,157.087
C02589=1052.678,293.038,-104.495,172.642,37.490,157.086
C02590=1052.672,292.790,-104.463,172.639,37.487,157.085
C02591=1052.666,292.542,-104.431,172.635,37.484,157.085
C02592=1052.659,292.295,-104.399,172.633,37.480,157.084
C02593=1052.652,292.047,-104.368,172.629,37.477,157.083
C02594=1052.646,291.799,-104.336,172.626,37.473,157.082
C02595=1052.639,291.551,-104.304,172.623,37.469,157.081
C02596=1052.633,291.303,-104.273,172.619,37.466,157.080
C02597=1052.626,291.055,-104.240,172.617,37.462,157.080
C02598=1052.620,290.797,-104.207,172.613,37.459,157.079
C02599=1052.613,290.538,-104.175,172.611,37.455,157.078
C02600=1052.606,290.279,-104.141,172.607,37.451,157.077
C02601=1052.599,290.020,-104.108,172.603,37.448,157.076
C02602=1052.593,289.773,-104.077,172.601,37.444,157.076
C02603=1052.587,289.524,-104.045,172.597,37.441,157.075
C02604=1052.580,289.276,-104.014,172.595,37.438,157.074
C02605=1052.573,289.028,-103.982,172.591,37.434,157.073
C02606=1052.566,288.781,-103.951,172.587,37.431,157.072
C02607=1052.561,288.533,-103.919,172.585,37.427,157.072
C02608=1052.554,288.285,-103.888,172.581,37.424,157.071
C02609=1052.548,288.037,-103.856,172.579,37.420,157.070
C02610=1052.541,287.789,-103.825,172.575,37.417,157.069
C02611=1052.534,287.541,-103.793,172.573,37.413,157.069
C02612=1052.528,287.293,-103.761,172.569,37.410,157.068
C02613=1052.521,287.045,-103.730,172.567,37.407,157.067
C02614=1052.515,286.797,-103.698,172.563,37.404,157.066
C02615=1052.509,286.550,-103.668,172.560,37.400,157.066
C02616=1052.502,286.302,-103.637,172.557,37.397,157.065
C02617=1052.495,286.054,-103.605,172.554,37.393,157.064
C02618=1052.489,285.806,-103.574,172.551,37.390,157.063
C02619=1052.482,285.558,-103.542,172.548,37.386,157.062
C02620=1052.476,285.309,-103.512,172.545,37.383,157.062
C02621=1052.469,285.062,-103.481,172.542,37.380,157.061
C02622=1052.463,284.814,-103.449,172.539,37.376,157.060
C02623=1052.456,284.566,-103.418,172.536,37.373,157.059
C02624=1052.450,284.318,-103.387,172.532,37.370,157.059
C02625=1052.443,284.070,-103.356,172.530,37.366,157.058
C02626=1052.437,283.823,-103.324,172.526,37.363,157.057
C02627=1052.430,283.574,-103.294,172.524,37.359,157.056
C02628=1052.424,283.326,-103.262,172.520,37.356,157.055
C02629=1052.417,283.079,-103.231,172.518,37.353,157.055
C02630=1052.411,282.831,-103.201,172.514,37.349,157.054
C02631=1052.404,282.583,-103.169,172.512,37.346,157.053
C02632=1052.398,282.335,-103.138,172.509,37.342,157.052
C02633=1052.391,282.086,-103.107,172.505,37.339,157.052
C02634=1052.385,281.839,-103.076,172.503,37.335,157.051
C02635=1052.379,281.591,-103.045,172.499,37.332,157.050
C02636=1052.372,281.343,-103.014,172.497,37.329,157.049
C02637=1052.366,281.096,-102.983,172.493,37.326,157.049
C02638=1052.359,280.847,-102.952,172.491,37.322,157.048
C02639=1052.353,280.599,-102.921,172.488,37.319,157.047
C02640=1052.346,280.351,-102.890,172.485,37.315,157.046
C02641=1052.340,280.103,-102.859,172.482,37.312,157.045
C02642=1052.334,279.855,-102.828,172.479,37.308,157.045
C02643=1052.327,279.608,-102.797,172.476,37.305,157.044
C02644=1052.321,279.359,-102.766,172.473,37.302,157.043
C02645=1052.315,279.111,-102.736,172.470,37.298,157.042
C02646=1052.308,278.863,-102.704,172.467,37.295,157.042
C02647=1052.302,278.615,-102.674,172.464,37.291,157.041
C02648=1052.295,278.367,-102.644,172.461,37.289,157.040
C02649=1052.288,278.119,-102.612,172.458,37.285,157.039
C02650=1052.282,277.871,-102.582,172.455,37.282,157.039
C02651=1052.276,277.624,-102.551,172.453,37.278,157.038
C02652=1052.269,277.376,-102.521,172.449,37.275,157.037
C02653=1052.263,277.128,-102.490,172.447,37.272,157.036
C02654=1052.257,276.880,-102.459,172.443,37.268,157.036
C02655=1052.250,276.632,-102.429,172.441,37.265,157.035
C02656=1052.243,276.384,-102.398,172.438,37.262,157.034
C02657=1052.237,276.137,-102.367,172.435,37.258,157.034
C02658=1052.230,275.888,-102.337,172.432,37.255,157.033
C02659=1052.224,275.641,-102.306,172.430,37.251,157.032
C02660=1052.218,275.393,-102.275,172.426,37.249,157.031
C02661=1052.212,275.145,-102.245,172.424,37.245,157.031
C02662=1052.205,274.897,-102.215,172.420,37.242,157.030
C02663=1052.199,274.649,-102.185,172.417,37.238,157.029
C02664=1052.193,274.400,-102.154,172.415,37.235,157.028
C02665=1052.185,274.153,-102.123,172.411,37.232,157.028
C02666=1052.179,273.905,-102.093,172.409,37.228,157.027
C02667=1052.173,273.656,-102.062,172.406,37.225,157.026
C02668=1052.166,273.409,-102.032,172.403,37.222,157.025
C02669=1052.160,273.160,-102.001,172.400,37.218,157.025
C02670=1052.154,272.913,-101.971,172.398,37.215,157.024
C02671=1052.147,272.664,-101.941,172.394,37.212,157.023
C02672=1052.141,272.416,-101.911,172.392,37.208,157.022
C02673=1052.135,272.168,-101.880,172.389,37.205,157.022
C02674=1052.128,271.920,-101.850,172.386,37.202,157.021
C02675=1052.122,271.672,-101.819,172.383,37.199,157.020
C02676=1052.115,271.424,-101.790,172.381,37.195,157.019
C02677=1052.109,271.176,-101.759,172.377,37.192,157.019
C02678=1052.102,270.928,-101.729,172.375,37.189,157.018
C02679=1052.096,270.680,-101.699,172.372,37.185,157.017
C02680=1052.090,270.432,-101.669,172.370,37.182,157.017
C02681=1052.083,270.183,-101.639,172.366,37.179,157.016
C02682=1052.077,269.936,-101.609,172.364,37.175,157.015
C02683=1052.070,269.687,-101.578,172.361,37.172,157.014
C02684=1052.064,269.440,-101.549,172.358,37.169,157.014
C02685=1052.057,269.191,-101.518,172.355,37.165,157.013
C02686=1052.051,268.944,-101.488,172.353,37.162,157.012
C02687=1052.044,268.694,-101.458,172.349,37.159,157.011
C02688=1052.038,268.447,-101.428,172.347,37.155,157.011
C02689=1052.032,268.198,-101.398,172.344,37.153,157.010
C02690=1052.025,267.951,-101.368,172.342,37.149,157.009
C02691=1052.018,267.702,-101.338,172.338,37.146,157.008
C02692=1052.012,267.454,-101.308,172.336,37.143,157.008
C02693=1052.006,267.207,-101.278,172.333,37.139,157.007
C02694=1051.999,266.958,-101.249,172.331,37.136,157.006
C02695=1051.993,266.710,-101.219,172.327,37.133,157.006
C02696=1051.986,266.462,-101.188,172.325,37.130,157.005
C02697=1051.980,266.213,-101.159,172.322,37.126,157.004
C02698=1051.973,265.965,-101.129,172.320,37.123,157.003
C02699=1051.967,265.718,-101.099,172.316,37.120,157.003
C02700=1051.961,265.469,-101.069,172.314,37.116,157.002
C02701=1051.954,265.221,-101.039,172.311,37.113,157.001
C02702=1051.948,264.973,-101.010,172.309,37.110,157.000
C02703=1051.942,264.725,-100.980,172.305,37.106,157.000
C02704=1051.935,264.477,-100.950,172.303,37.104,156.999
C02705=1051.929,264.229,-100.921,172.300,37.100,156.998
C02706=1051.922,263.983,-100.891,172.298,37.097,156.998
C02707=1051.916,263.737,-100.861,172.295,37.094,156.997
C02708=1051.909,263.492,-100.832,172.292,37.090,156.996
C02709=1051.904,263.246,-100.803,172.289,37.087,156.995
C02710=1051.897,263.000,-100.774,172.287,37.084,156.995
C02711=1051.891,262.754,-100.744,172.284,37.081,156.994
C02712=1051.884,262.509,-100.714,172.282,37.077,156.993
C02713=1051.878,262.263,-100.686,172.278,37.074,156.993
C02714=1051.871,262.015,-100.656,172.276,37.071,156.992
C02715=1051.864,261.766,-100.627,172.274,37.068,156.991
C02716=1051.858,261.518,-100.597,172.271,37.065,156.991
C02717=1051.852,261.271,-100.568,172.268,37.061,156.990
C02718=1051.845,261.022,-100.538,172.265,37.059,156.989
C02719=1051.838,260.774,-100.509,172.263,37.055,156.988
C02720=1051.832,260.526,-100.480,172.260,37.052,156.988
C02721=1051.825,260.277,-100.450,172.258,37.049,156.987
C02722=1051.819,260.029,-100.421,172.254,37.046,156.986
C02723=1051.813,259.781,-100.392,172.252,37.042,156.986
C02724=1051.805,259.533,-100.362,172.249,37.039,156.985
C02725=1051.799,259.285,-100.333,172.247,37.036,156.984
C02726=1051.793,259.037,-100.304,172.244,37.033,156.984
C02727=1051.785,258.788,-100.275,172.241,37.029,156.983
C02728=1051.779,258.540,-100.246,172.238,37.026,156.982
C02729=1051.772,258.292,-100.216,172.236,37.023,156.981
C02730=1051.766,258.044,-100.187,172.233,37.020,156.981
C02731=1051.759,257.795,-100.158,172.231,37.016,156.980
C02732=1051.753,257.547,-100.129,172.228,37.013,156.979
C02733=1051.747,257.299,-100.100,172.225,37.010,156.979
C02734=1051.741,257.051,-100.071,172.223,37.007,156.978
C02735=1051.734,256.802,-100.041,172.220,37.004,156.977
C02736=1051.727,256.555,-100.011,172.218,37.000,156.976
C02737=1051.721,256.307,-99.982,172.215,36.998,156.976
C02738=1051.715,256.058,-99.953,172.213,36.994,156.975
C02739=1051.708,255.810,-99.924,172.210,36.991,156.974
C02740=1051.702,255.561,-99.895,172.207,36.988,156.974
C02741=1051.695,255.313,-99.866,172.204,36.985,156.973
C02742=1051.689,255.065,-99.837,172.202,36.981,156.972
C02743=1051.682,254.817,-99.808,172.199,36.978,156.972
C02744=1051.675,254.569,-99.779,172.197,36.975,156.971
C02745=1051.669,254.320,-99.750,172.194,36.971,156.970
C02746=1051.663,254.072,-99.721,172.192,36.968,156.969
C02747=1051.657,253.824,-99.692,172.189,36.965,156.969
C02748=1051.650,253.576,-99.663,172.187,36.962,156.968
C02749=1051.644,253.328,-99.634,172.184,36.958,156.967
C02750=1051.638,253.080,-99.605,172.181,36.955,156.967
C02751=1051.631,252.830,-99.576,172.179,36.952,156.966
C02752=1051.625,252.582,-99.547,172.176,36.949,156.965
C02753=1051.619,252.334,-99.518,172.174,36.945,156.964
C02754=1051.612,252.086,-99.490,172.171,36.942,156.964
C02755=1051.606,251.838,-99.461,172.169,36.939,156.963
C02756=1051.599,251.590,-99.431,172.166,36.936,156.962
C02757=1051.593,251.342,-99.402,172.164,36.932,156.962
C02758=1051.587,251.094,-99.373,172.161,36.929,156.961
C02759=1051.581,250.845,-99.345,172.159,36.926,156.960
C02760=1051.575,250.597,-99.316,172.156,36.923,156.960
C02761=1051.568,250.348,-99.287,172.154,36.919,156.959
C02762=1051.562,250.102,-99.258,172.151,36.916,156.958
C02763=1051.555,249.855,-99.230,172.149,36.913,156.957
C02764=1051.549,249.609,-99.201,172.147,36.909,156.957
C02765=1051.543,249.362,-99.172,172.143,36.906,156.956
C02766=1051.537,249.115,-99.144,172.141,36.903,156.955
C02767=1051.530,248.869,-99.115,172.138,36.900,156.955
C02768=1051.523,248.623,-99.087,172.136,36.896,156.954
C02769=1051.518,248.376,-99.058,172.133,36.893,156.953
C02770=1051.511,248.128,-99.030,172.131,36.890,156.953
C02771=1051.505,247.880,-99.001,172.128,36.887,156.952
C02772=1051.499,247.631,-98.973,172.126,36.883,156.951
C02773=1051.493,247.383,-98.943,172.123,36.880,156.950
C02774=1051.487,247.135,-98.914,172.121,36.877,156.950
C02775=1051.481,246.886,-98.886,172.118,36.873,156.949
C02776=1051.474,246.638,-98.857,172.116,36.870,156.948
C02777=1051.468,246.390,-98.829,172.114,36.867,156.948
C02778=1051.462,246.141,-98.800,172.111,36.863,156.947
C02779=1051.455,245.893,-98.771,172.109,36.860,156.946
C02780=1051.449,245.645,-98.743,172.106,36.857,156.945
C02781=1051.442,245.397,-98.714,172.104,36.854,156.945
C02782=1051.436,245.148,-98.686,172.101,36.850,156.944
C02783=1051.430,244.900,-98.657,172.099,36.847,156.943
C02784=1051.423,244.651,-98.629,172.096,36.844,156.943
C02785=1051.417,244.403,-98.600,172.094,36.841,156.942
C02786=1051.411,244.155,-98.573,172.091,36.837,156.941
C02787=1051.405,243.906,-98.544,172.089,36.834,156.941
C02788=1051.398,243.658,-98.515,172.087,36.831,156.940
C02789=1051.392,243.409,-98.488,172.084,36.828,156.939
C02790=1051.385,243.161,-98.458,172.083,36.824,156.938
C02791=1051.379,242.913,-98.431,172.080,36.821,156.938
C02792=1051.373,242.664,-98.402,172.078,36.818,156.937
C02793=1051.366,242.416,-98.374,172.075,36.815,156.936
C02794=1051.360,242.168,-98.346,172.073,36.811,156.936
C02795=1051.354,241.920,-98.317,172.071,36.808,156.935
C02796=1051.348,241.672,-98.289,172.068,36.805,156.934
C02797=1051.342,241.423,-98.261,172.066,36.802,156.934
C02798=1051.335,241.175,-98.233,172.063,36.798,156.933
C02799=1051.328,240.927,-98.205,172.061,36.795,156.932
C02800=1051.322,240.678,-98.176,172.058,36.792,156.931
C02801=1051.315,240.429,-98.149,172.056,36.789,156.931
C02802=1051.309,240.181,-98.121,172.053,36.785,156.930
C02803=1051.302,239.933,-98.092,172.051,36.782,156.929
C02804=1051.296,239.684,-98.064,172.048,36.779,156.929
C02805=1051.289,239.436,-98.036,172.046,36.776,156.928
C02806=1051.283,239.187,-98.008,172.044,36.773,156.927
C02807=1051.277,238.940,-97.981,172.041,36.769,156.927
C02808=1051.271,238.691,-97.952,172.039,36.766,156.926
C02809=1051.264,238.443,-97.924,172.036,36.763,156.925
C02810=1051.257,238.195,-97.896,172.034,36.760,156.925
C02811=1051.251,237.946,-97.869,172.032,36.756,156.924
C02812=1051.245,237.697,-97.840,172.030,36.753,156.923
C02813=1051.238,237.449,-97.812,172.028,36.750,156.922
C02814=1051.232,237.201,-97.785,172.025,36.747,156.922
C02815=1051.226,236.952,-97.757,172.023,36.743,156.921
C02816=1051.219,236.704,-97.729,172.020,36.740,156.920
C02817=1051.212,236.456,-97.701,172.018,36.737,156.920
C02818=1051.206,236.208,-97.673,172.015,36.734,156.919
C02819=1051.200,235.959,-97.645,172.013,36.730,156.918
C02820=1051.194,235.711,-97.617,172.011,36.727,156.918
C02821=1051.187,235.463,-97.589,172.008,36.724,156.917
C02822=1051.180,235.211,-97.562,172.007,36.721,156.916
C02823=1051.174,234.961,-97.534,172.004,36.717,156.916
C02824=1051.168,234.710,-97.505,172.002,36.714,156.915
C02825=1051.162,234.459,-97.477,171.999,36.711,156.914
C02826=1051.155,234.210,-97.450,171.997,36.708,156.914
C02827=1051.149,233.963,-97.422,171.994,36.704,156.913
C02828=1051.143,233.714,-97.394,171.992,36.701,156.912
C02829=1051.136,233.465,-97.366,171.990,36.697,156.911
C02830=1051.130,233.217,-97.338,171.988,36.695,156.911
C02831=1051.123,232.969,-97.311,171.986,36.691,156.910
C02832=1051.117,232.721,-97.283,171.983,36.688,156.909
C02833=1051.111,232.472,-97.255,171.981,36.684,156.909
C02834=1051.104,232.223,-97.227,171.979,36.681,156.908
C02835=1051.098,231.975,-97.201,171.976,36.678,156.907
C02836=1051.092,231.727,-97.173,171.974,36.675,156.907
C02837=1051.085,231.478,-97.145,171.972,36.671,156.906
C02838=1051.078,231.230,-97.117,171.970,36.668,156.905
C02839=1051.072,230.982,-97.090,171.967,36.665,156.904
C02840=1051.066,230.733,-97.063,171.965,36.662,156.904
C02841=1051.060,230.484,-97.035,171.962,36.658,156.903
C02842=1051.054,230.237,-97.007,171.960,36.655,156.902
C02843=1051.047,229.988,-96.980,171.959,36.652,156.902
C02844=1051.041,229.739,-96.953,171.956,36.649,156.901
C02845=1051.034,229.491,-96.925,171.954,36.645,156.900
C02846=1051.028,229.243,-96.898,171.951,36.642,156.900
C02847=1051.021,228.994,-96.870,171.949,36.639,156.899
C02848=1051.015,228.745,-96.843,171.947,36.636,156.898
C02849=1051.009,228.498,-96.815,171.945,36.632,156.898
C02850=1051.003,228.249,-96.788,171.943,36.629,156.897
C02851=1050.996,228.000,-96.761,171.940,36.626,156.896
C02852=1050.990,227.752,-96.733,171.938,36.623,156.896
C02853=1050.983,227.503,-96.706,171.935,36.619,156.895
C02854=1050.976,227.255,-96.679,171.934,36.616,156.894
C02855=1050.970,227.006,-96.652,171.932,36.612,156.893
C02856=1050.964,226.758,-96.625,171.929,36.609,156.893
C02857=1050.957,226.510,-96.597,171.927,36.606,156.892
C02858=1050.950,226.261,-96.570,171.924,36.603,156.891
C02859=1050.944,226.013,-96.543,171.923,36.600,156.891
C02860=1050.938,225.764,-96.516,171.920,36.596,156.890
C02861=1050.931,225.516,-96.488,171.918,36.593,156.889
C02862=1050.925,225.268,-96.462,171.916,36.590,156.889
C02863=1050.918,225.019,-96.434,171.913,36.587,156.888
C02864=1050.912,224.771,-96.408,171.912,36.583,156.887
C02865=1050.906,224.522,-96.380,171.909,36.580,156.887
C02866=1050.899,224.273,-96.353,171.907,36.577,156.886
C02867=1050.894,224.025,-96.326,171.905,36.573,156.885
C02868=1050.887,223.776,-96.298,171.903,36.570,156.885
C02869=1050.881,223.528,-96.272,171.901,36.567,156.884
C02870=1050.874,223.280,-96.245,171.898,36.564,156.883
C02871=1050.867,223.031,-96.218,171.896,36.560,156.882
C02872=1050.861,222.783,-96.190,171.894,36.557,156.882
C02873=1050.855,222.534,-96.163,171.892,36.553,156.881
C02874=1050.849,222.286,-96.137,171.890,36.550,156.880
C02875=1050.842,222.037,-96.109,171.887,36.547,156.880
C02876=1050.836,221.789,-96.083,171.886,36.544,156.879
C02877=1050.829,221.540,-96.056,171.883,36.540,156.878
C02878=1050.823,221.282,-96.027,171.881,36.537,156.878
C02879=1050.817,221.024,-96.000,171.878,36.533,156.877
C02880=1050.810,220.765,-95.972,171.877,36.530,156.876
C02881=1050.804,220.507,-95.943,171.875,36.527,156.875
C02882=1050.796,220.259,-95.916,171.872,36.523,156.875
C02883=1050.791,220.011,-95.890,171.870,36.520,156.874
C02884=1050.784,219.761,-95.863,171.868,36.516,156.873
C02885=1050.777,219.513,-95.836,171.866,36.513,156.873
C02886=1050.771,219.264,-95.810,171.864,36.510,156.872
C02887=1050.764,219.016,-95.782,171.861,36.507,156.871
C02888=1050.758,218.768,-95.756,171.860,36.503,156.871
C02889=1050.752,218.519,-95.729,171.857,36.500,156.870
C02890=1050.745,218.271,-95.703,171.855,36.497,156.869
C02891=1050.739,218.022,-95.676,171.854,36.494,156.869
C02892=1050.732,217.774,-95.650,171.851,36.490,156.868
C02893=1050.726,217.525,-95.622,171.849,36.487,156.867
C02894=1050.719,217.277,-95.596,171.846,36.483,156.867
C02895=1050.713,217.028,-95.569,171.845,36.480,156.866
C02896=1050.707,216.780,-95.542,171.843,36.477,156.865
C02897=1050.700,216.531,-95.516,171.840,36.474,156.865
C02898=1050.694,216.283,-95.489,171.839,36.470,156.864
C02899=1050.687,216.034,-95.463,171.836,36.467,156.863
C02900=1050.681,215.786,-95.436,171.834,36.464,156.862
C02901=1050.674,215.537,-95.410,171.832,36.460,156.862
C02902=1050.668,215.288,-95.383,171.830,36.457,156.861
C02903=1050.663,215.040,-95.356,171.828,36.454,156.860
C02904=1050.655,214.791,-95.330,171.826,36.451,156.860
C02905=1050.650,214.543,-95.303,171.824,36.447,156.859
C02906=1050.643,214.294,-95.277,171.822,36.444,156.858
C02907=1050.637,214.046,-95.250,171.820,36.440,156.858
C02908=1050.630,213.797,-95.224,171.818,36.437,156.857
C02909=1050.624,213.549,-95.197,171.815,36.434,156.856
C02910=1050.617,213.301,-95.171,171.814,36.430,156.855
C02911=1050.611,213.052,-95.144,171.811,36.427,156.855
C02912=1050.604,212.804,-95.118,171.809,36.424,156.854
C02913=1050.598,212.554,-95.091,171.808,36.420,156.853
C02914=1050.592,212.306,-95.064,171.805,36.417,156.853
C02915=1050.586,212.058,-95.038,171.804,36.413,156.852
C02916=1050.579,211.809,-95.012,171.801,36.410,156.851
C02917=1050.573,211.561,-94.985,171.799,36.407,156.851
C02918=1050.566,211.312,-94.959,171.798,36.403,156.850
C02919=1050.560,211.063,-94.933,171.795,36.400,156.849
C02920=1050.554,210.815,-94.907,171.793,36.397,156.849
C02921=1050.547,210.566,-94.880,171.791,36.393,156.848
C02922=1050.541,210.318,-94.854,171.789,36.390,156.847
C02923=1050.534,210.070,-94.828,171.788,36.386,156.846
C02924=1050.528,209.821,-94.802,171.785,36.383,156.846
C02925=1050.522,209.572,-94.775,171.783,36.380,156.845
C02926=1050.515,209.324,-94.749,171.781,36.376,156.844
C02927=1050.508,209.076,-94.723,171.779,36.373,156.844
C02928=1050.503,208.827,-94.697,171.778,36.370,156.843
C02929=1050.496,208.578,-94.671,171.775,36.367,156.842
C02930=1050.489,208.330,-94.644,171.773,36.363,156.842
C02931=1050.483,208.082,-94.618,171.771,36.359,156.841
C02932=1050.477,207.832,-94.592,171.769,36.356,156.840
C02933=1050.470,207.584,-94.566,171.768,36.353,156.840
C02934=1050.464,207.331,-94.539,171.765,36.349,156.839
C02935=1050.457,207.078,-94.513,171.763,36.346,156.838
C02936=1050.450,206.825,-94.487,171.761,36.343,156.837
C02937=1050.444,206.572,-94.460,171.759,36.339,156.837
C02938=1050.418,205.521,-94.354,171.530,36.243,156.818
C02939=1050.412,205.272,-94.329,171.527,36.240,156.817
C02940=1050.406,205.023,-94.304,171.525,36.238,156.816
C02941=1050.400,204.774,-94.279,171.522,36.235,156.816
C02942=1050.394,204.526,-94.254,171.520,36.233,156.815
C02943=1050.388,204.277,-94.229,171.517,36.230,156.815
C02944=1050.382,204.028,-94.204,171.515,36.228,156.814
C02945=1050.376,203.780,-94.179,171.512,36.225,156.814
C02946=1050.369,203.531,-94.155,171.509,36.223,156.813
C02947=1050.364,203.283,-94.130,171.507,36.220,156.813
C02948=1050.358,203.034,-94.104,171.504,36.217,156.812
C02949=1050.352,202.785,-94.080,171.502,36.215,156.812
C02950=1050.346,202.537,-94.055,171.499,36.212,156.811
C02951=1050.340,202.288,-94.030,171.497,36.210,156.811
C02952=1050.334,202.039,-94.005,171.494,36.207,156.810
C02953=1050.328,201.790,-93.979,171.492,36.205,156.810
C02954=1050.322,201.542,-93.955,171.489,36.202,156.809
C02955=1050.315,201.293,-93.930,171.486,36.200,156.809
C02956=1050.310,201.044,-93.906,171.484,36.197,156.808
C02957=1050.303,200.795,-93.881,171.482,36.195,156.808
C02958=1050.297,200.547,-93.857,171.479,36.192,156.807
C02959=1050.291,200.298,-93.832,171.476,36.190,156.807
C02960=1050.284,200.049,-93.807,171.474,36.187,156.806
C02961=1050.279,199.800,-93.783,171.472,36.185,156.806
C02962=1050.273,199.552,-93.758,171.469,36.183,156.805
C02963=1050.266,199.303,-93.734,171.466,36.180,156.805
C02964=1050.260,199.055,-93.709,171.464,36.178,156.804
C02965=1050.254,198.806,-93.685,171.461,36.175,156.804
C02966=1050.248,198.557,-93.660,171.459,36.173,156.804
C02967=1050.241,198.309,-93.636,171.456,36.171,156.803
C02968=1050.235,198.059,-93.611,171.454,36.168,156.803
C02969=1050.230,197.811,-93.587,171.452,36.166,156.802
C02970=1050.223,197.562,-93.562,171.449,36.164,156.802
C02971=1050.217,197.313,-93.537,171.446,36.161,156.801
C02972=1050.211,197.065,-93.514,171.444,36.159,156.801
C02973=1050.205,196.816,-93.488,171.442,36.156,156.800
C02974=1050.198,196.567,-93.464,171.438,36.154,156.800
C02975=1050.193,196.319,-93.440,171.436,36.151,156.799
C02976=1050.187,196.069,-93.415,171.434,36.149,156.799
C02977=1050.181,195.822,-93.391,171.432,36.147,156.798
C02978=1050.175,195.572,-93.366,171.429,36.144,156.798
C02979=1050.168,195.323,-93.342,171.426,36.142,156.797
C02980=1050.163,195.075,-93.318,171.424,36.139,156.797
C02981=1050.156,194.826,-93.293,171.422,36.137,156.796
C02982=1050.151,194.578,-93.269,171.419,36.134,156.796
C02983=1050.144,194.329,-93.245,171.417,36.132,156.795
C02984=1050.138,194.080,-93.220,171.414,36.129,156.795
C02985=1050.133,193.831,-93.196,171.412,36.128,156.794
C02986=1050.126,193.582,-93.172,171.409,36.125,156.794
C02987=1050.121,193.334,-93.147,171.407,36.123,156.794
C02988=1050.114,193.085,-93.123,171.405,36.120,156.793
C02989=1050.109,192.836,-93.099,171.402,36.118,156.793
C02990=1050.102,192.588,-93.075,171.399,36.115,156.792
C02991=1050.097,192.339,-93.051,171.397,36.113,156.792
C02992=1050.090,192.090,-93.027,171.395,36.110,156.791
C02993=1050.084,191.841,-93.002,171.393,36.108,156.791
C02994=1050.078,191.592,-92.978,171.390,36.106,156.790
C02995=1050.072,191.343,-92.954,171.387,36.103,156.790
C02996=1050.066,191.095,-92.930,171.385,36.101,156.789
C02997=1050.060,190.846,-92.905,171.383,36.099,156.789
C02998=1050.054,190.598,-92.881,171.380,36.096,156.788
C02999=1050.047,190.313,-92.854,171.378,36.093,156.788
C03000=1050.041,190.029,-92.826,171.375,36.091,156.787
C03001=1050.034,189.744,-92.798,171.373,36.088,156.787
C03002=1050.027,189.460,-92.771,171.369,36.085,156.786
C03003=1050.021,189.211,-92.747,171.367,36.083,156.786
C03004=1050.015,188.963,-92.723,171.365,36.081,156.785
C03005=1050.009,188.714,-92.699,171.362,36.078,156.785
C03006=1050.004,188.465,-92.674,171.360,36.076,156.784
C03007=1049.997,188.217,-92.651,171.358,36.074,156.784
C03008=1049.992,187.968,-92.626,171.355,36.071,156.783
C03009=1049.986,187.719,-92.602,171.353,36.069,156.783
C03010=1049.980,187.470,-92.578,171.350,36.066,156.782
C03011=1049.974,187.222,-92.554,171.348,36.064,156.782
C03012=1049.968,186.972,-92.530,171.346,36.062,156.781
C03013=1049.962,186.723,-92.507,171.344,36.060,156.781
C03014=1049.957,186.475,-92.482,171.341,36.057,156.781
C03015=1049.950,186.226,-92.458,171.339,36.055,156.780
C03016=1049.945,185.977,-92.434,171.337,36.052,156.780
C03017=1049.939,185.729,-92.410,171.335,36.050,156.779
C03018=1049.933,185.479,-92.387,171.331,36.047,156.779
C03019=1049.927,185.231,-92.363,171.329,36.045,156.778
C03020=1049.921,184.983,-92.339,171.327,36.043,156.778
C03021=1049.915,184.733,-92.315,171.325,36.041,156.777
C03022=1049.909,184.485,-92.291,171.322,36.038,156.777
C03023=1049.904,184.235,-92.267,171.320,36.036,156.776
C03024=1049.897,183.987,-92.243,171.318,36.033,156.776
C03025=1049.891,183.739,-92.220,171.316,36.031,156.776
C03026=1049.885,183.489,-92.196,171.313,36.029,156.775
C03027=1049.879,183.241,-92.173,171.311,36.027,156.775
C03028=1049.872,182.992,-92.149,171.308,36.025,156.774
C03029=1049.867,182.743,-92.126,171.306,36.023,156.774
C03030=1049.860,182.494,-92.102,171.304,36.020,156.773
C03031=1049.854,182.245,-92.079,171.301,36.018,156.773
C03032=1049.848,181.997,-92.055,171.299,36.016,156.773
C03033=1049.842,181.748,-92.031,171.297,36.014,156.772
C03034=1049.836,181.499,-92.008,171.295,36.012,156.772
C03035=1049.829,181.250,-91.984,171.292,36.009,156.771
C03036=1049.824,181.001,-91.961,171.290,36.008,156.771
C03037=1049.817,180.753,-91.938,171.287,36.005,156.770
C03038=1049.810,180.503,-91.915,171.285,36.003,156.770
C03039=1049.804,180.255,-91.891,171.283,36.001,156.770
C03040=1049.798,180.005,-91.868,171.280,35.999,156.769
C03041=1049.792,179.757,-91.844,171.278,35.996,156.769
C03042=1049.786,179.508,-91.821,171.276,35.995,156.768
C03043=1049.780,179.259,-91.797,171.274,35.992,156.768
C03044=1049.774,179.010,-91.774,171.272,35.990,156.768
C03045=1049.768,178.762,-91.751,171.269,35.988,156.767
C03046=1049.762,178.513,-91.727,171.267,35.986,156.767
C03047=1049.756,178.264,-91.704,171.265,35.984,156.766
C03048=1049.750,178.015,-91.681,171.263,35.982,156.766
C03049=1049.743,177.766,-91.658,171.260,35.979,156.765
C03050=1049.737,177.518,-91.634,171.258,35.977,156.765
C03051=1049.731,177.269,-91.611,171.255,35.975,156.765
C03052=1049.725,177.019,-91.588,171.253,35.972,156.764
C03053=1049.719,176.771,-91.564,171.251,35.971,156.764
C03054=1049.713,176.522,-91.541,171.248,35.968,156.763
C03055=1049.707,176.273,-91.518,171.246,35.966,156.763
C03056=1049.700,176.024,-91.494,171.244,35.964,156.762
C03057=1049.695,175.775,-91.471,171.242,35.962,156.762
C03058=1049.688,175.527,-91.449,171.239,35.959,156.762
C03059=1049.682,175.279,-91.425,171.237,35.958,156.761
C03060=1049.676,175.029,-91.402,171.235,35.955,156.761
C03061=1049.670,174.780,-91.379,171.233,35.953,156.760
C03062=1049.664,174.532,-91.356,171.231,35.951,156.760
C03063=1049.657,174.247,-91.330,171.228,35.948,156.759
C03064=1049.651,173.962,-91.303,171.225,35.946,156.759
C03065=1049.643,173.677,-91.276,171.223,35.943,156.758
C03066=1049.637,173.393,-91.250,171.221,35.941,156.758
C03067=1049.631,173.144,-91.227,171.218,35.939,156.758
C03068=1049.624,172.895,-91.203,171.216,35.937,156.757
C03069=1049.618,172.646,-91.180,171.214,35.935,156.757
C03070=1049.613,172.397,-91.157,171.212,35.932,156.756
C03071=1049.606,172.148,-91.135,171.210,35.930,156.756
C03072=1049.601,171.899,-91.112,171.207,35.928,156.755
C03073=1049.594,171.650,-91.088,171.205,35.926,156.755
C03074=1049.588,171.401,-91.065,171.203,35.924,156.755
C03075=1049.582,171.153,-91.042,171.201,35.922,156.754
C03076=1049.577,170.904,-91.019,171.199,35.920,156.754
C03077=1049.570,170.655,-90.997,171.196,35.918,156.753
C03078=1049.565,170.406,-90.974,171.194,35.916,156.753
C03079=1049.559,170.157,-90.951,171.192,35.913,156.753
C03080=1049.552,169.908,-90.927,171.190,35.911,156.752
C03081=1049.546,169.659,-90.904,171.188,35.909,156.752
C03082=1049.541,169.411,-90.881,171.185,35.907,156.751
C03083=1049.534,169.162,-90.859,171.183,35.905,156.751
C03084=1049.529,168.913,-90.836,171.181,35.903,156.751
C03085=1049.523,168.664,-90.813,171.179,35.900,156.750
C03086=1049.517,168.415,-90.790,171.176,35.898,156.750
C03087=1049.511,168.166,-90.767,171.174,35.896,156.749
C03088=1049.506,167.917,-90.744,171.172,35.894,156.749
C03089=1049.499,167.669,-90.722,171.170,35.892,156.748
C03090=1049.493,167.419,-90.698,171.168,35.890,156.748
C03091=1049.487,167.170,-90.675,171.165,35.887,156.748
C03092=1049.481,166.921,-90.652,171.163,35.885,156.747
C03093=1049.476,166.673,-90.629,171.161,35.883,156.747
C03094=1049.469,166.424,-90.607,171.159,35.881,156.746
C03095=1049.463,166.175,-90.584,171.157,35.879,156.746
C03096=1049.458,165.926,-90.561,171.155,35.877,156.746
C03097=1049.452,165.677,-90.538,171.153,35.874,156.745
C03098=1049.446,165.428,-90.515,171.151,35.872,156.745
C03099=1049.440,165.180,-90.493,171.149,35.871,156.744
C03100=1049.434,164.931,-90.470,171.147,35.868,156.744
C03101=1049.429,164.681,-90.448,171.144,35.866,156.744
C03102=1049.423,164.433,-90.425,171.142,35.864,156.743
C03103=1049.416,164.184,-90.402,171.140,35.862,156.743
C03104=1049.411,163.935,-90.380,171.138,35.859,156.742
C03105=1049.405,163.686,-90.357,171.136,35.858,156.742
C03106=1049.399,163.437,-90.334,171.133,35.855,156.741
C03107=1049.393,163.188,-90.311,171.131,35.853,156.741
C03108=1049.387,162.940,-90.288,171.129,35.851,156.741
C03109=1049.382,162.690,-90.266,171.128,35.849,156.740
C03110=1049.376,162.441,-90.243,171.126,35.846,156.740
C03111=1049.370,162.192,-90.220,171.123,35.845,156.739
C03112=1049.364,161.944,-90.198,171.121,35.842,156.739
C03113=1049.358,161.695,-90.175,171.119,35.840,156.739
C03114=1049.353,161.446,-90.153,171.117,35.838,156.738
C03115=1049.347,161.197,-90.130,171.115,35.836,156.738
C03116=1049.341,160.949,-90.108,171.112,35.833,156.737
C03117=1049.335,160.700,-90.085,171.110,35.831,156.737
C03118=1049.330,160.450,-90.063,171.108,35.830,156.737
C03119=1049.323,160.202,-90.040,171.107,35.827,156.736
C03120=1049.318,159.953,-90.017,171.105,35.825,156.736
C03121=1049.311,159.704,-89.996,171.102,35.823,156.735
C03122=1049.305,159.455,-89.973,171.100,35.822,156.735
C03123=1049.299,159.206,-89.950,171.098,35.819,156.735
C03124=1049.293,158.957,-89.929,171.096,35.817,156.734
C03125=1049.287,158.708,-89.906,171.094,35.815,156.734
C03126=1049.281,158.459,-89.884,171.091,35.813,156.734
C03127=1049.274,158.174,-89.858,171.089,35.811,156.733
C03128=1049.267,157.889,-89.833,171.087,35.809,156.733
C03129=1049.260,157.603,-89.807,171.085,35.806,156.732
C03130=1049.253,157.318,-89.782,171.082,35.804,156.732
C03131=1049.247,157.069,-89.759,171.080,35.802,156.731
C03132=1049.241,156.820,-89.738,171.078,35.800,156.731
C03133=1049.235,156.572,-89.715,171.076,35.798,156.731
C03134=1049.229,156.322,-89.693,171.074,35.796,156.730
C03135=1049.223,156.074,-89.671,171.072,35.794,156.730
C03136=1049.217,155.824,-89.648,171.069,35.792,156.729
C03137=1049.211,155.575,-89.626,171.067,35.790,156.729
C03138=1049.205,155.326,-89.604,171.065,35.788,156.729
C03139=1049.200,155.078,-89.582,171.063,35.786,156.728
C03140=1049.193,154.829,-89.560,171.062,35.784,156.728
C03141=1049.187,154.580,-89.538,171.060,35.782,156.728
C03142=1049.181,154.331,-89.516,171.057,35.780,156.727
C03143=1049.175,154.081,-89.494,171.055,35.777,156.727
C03144=1049.169,153.833,-89.472,171.053,35.776,156.726
C03145=1049.163,153.584,-89.450,171.051,35.774,156.726
C03146=1049.156,153.335,-89.428,171.049,35.772,156.726
C03147=1049.151,153.086,-89.405,171.047,35.770,156.725
C03148=1049.145,152.836,-89.384,171.045,35.767,156.725
C03149=1049.139,152.589,-89.362,171.043,35.766,156.724
C03150=1049.133,152.339,-89.340,171.041,35.764,156.724
C03151=1049.126,152.091,-89.318,171.039,35.762,156.724
C03152=1049.121,151.841,-89.296,171.037,35.760,156.723
C03153=1049.115,151.592,-89.274,171.034,35.758,156.723
C03154=1049.108,151.343,-89.252,171.032,35.756,156.723
C03155=1049.102,151.094,-89.230,171.031,35.754,156.722
C03156=1049.097,150.845,-89.208,171.029,35.752,156.722
C03157=1049.091,150.596,-89.186,171.027,35.750,156.722
C03158=1049.084,150.348,-89.164,171.025,35.748,156.721
C03159=1049.078,150.098,-89.142,171.022,35.746,156.721
C03160=1049.072,149.849,-89.121,171.020,35.744,156.720
C03161=1049.066,149.601,-89.098,171.018,35.742,156.720
C03162=1049.061,149.352,-89.077,171.017,35.740,156.720
C03163=1049.055,149.103,-89.055,171.015,35.738,156.719
C03164=1049.049,148.853,-89.033,171.012,35.736,156.719
C03165=1049.042,148.604,-89.012,171.010,35.734,156.718
C03166=1049.036,148.356,-88.989,171.008,35.732,156.718
C03167=1049.030,148.107,-88.968,171.006,35.730,156.718
C03168=1049.024,147.858,-88.946,171.005,35.728,156.717
C03169=1049.018,147.609,-88.925,171.003,35.726,156.717
C03170=1049.013,147.359,-88.903,171.000,35.724,156.717
C03171=1049.006,147.111,-88.880,170.998,35.722,156.716
C03172=1049.001,146.862,-88.859,170.996,35.720,156.716
C03173=1048.994,146.613,-88.838,170.994,35.718,156.716
C03174=1048.987,146.364,-88.816,170.993,35.716,156.715
C03175=1048.981,146.115,-88.795,170.991,35.714,156.715
C03176=1048.975,145.866,-88.773,170.988,35.713,156.715
C03177=1048.970,145.617,-88.752,170.986,35.711,156.714
C03178=1048.963,145.368,-88.730,170.984,35.709,156.714
C03179=1048.957,145.119,-88.708,170.982,35.707,156.713
C03180=1048.951,144.869,-88.687,170.981,35.705,156.713
C03181=1048.946,144.621,-88.666,170.979,35.703,156.713
C03182=1048.939,144.372,-88.644,170.976,35.701,156.712
C03183=1048.933,144.123,-88.622,170.974,35.699,156.712
C03184=1048.927,143.874,-88.600,170.972,35.697,156.712
C03185=1048.921,143.625,-88.579,170.971,35.695,156.711
C03186=1048.915,143.376,-88.557,170.969,35.693,156.711
C03187=1048.909,143.127,-88.535,170.967,35.691,156.711
C03188=1048.903,142.878,-88.514,170.964,35.689,156.710
C03189=1048.897,142.629,-88.492,170.962,35.688,156.710
C03190=1048.891,142.379,-88.472,170.960,35.686,156.709
C03191=1048.884,142.095,-88.447,170.958,35.683,156.709
C03192=1048.877,141.809,-88.422,170.956,35.681,156.709
C03193=1048.871,141.523,-88.398,170.953,35.679,156.708
C03194=1048.863,141.238,-88.373,170.951,35.676,156.708
C03195=1048.857,140.989,-88.352,170.949,35.674,156.707
C03196=1048.851,140.740,-88.330,170.948,35.673,156.707
C03197=1048.845,140.492,-88.309,170.946,35.671,156.707
C03198=1048.839,140.242,-88.288,170.944,35.669,156.706
C03199=1048.833,139.992,-88.266,170.941,35.667,156.706
C03200=1048.827,139.743,-88.245,170.939,35.665,156.706
C03201=1048.822,139.495,-88.223,170.938,35.663,156.705
C03202=1048.815,139.246,-88.202,170.936,35.661,156.705
C03203=1048.808,138.997,-88.181,170.934,35.659,156.705
C03204=1048.803,138.748,-88.160,170.932,35.658,156.704
C03205=1048.797,138.498,-88.138,170.930,35.656,156.704
C03206=1048.790,138.249,-88.117,170.928,35.654,156.704
C03207=1048.785,138.001,-88.096,170.926,35.652,156.703
C03208=1048.778,137.752,-88.074,170.924,35.649,156.703
C03209=1048.773,137.502,-88.054,170.922,35.648,156.702
C03210=1048.767,137.253,-88.032,170.921,35.646,156.702
C03211=1048.760,137.005,-88.011,170.918,35.644,156.702
C03212=1048.754,136.755,-87.990,170.916,35.642,156.701
C03213=1048.749,136.506,-87.969,170.914,35.640,156.701
C03214=1048.742,136.257,-87.948,170.912,35.638,156.701
C03215=1048.736,136.009,-87.927,170.911,35.636,156.700
C03216=1048.730,135.760,-87.905,170.909,35.634,156.700
C03217=1048.723,135.510,-87.885,170.907,35.633,156.700
C03218=1048.718,135.262,-87.863,170.904,35.631,156.699
C03219=1048.712,135.012,-87.842,170.903,35.629,156.699
C03220=1048.705,134.763,-87.822,170.901,35.627,156.699
C03221=1048.700,134.514,-87.800,170.899,35.625,156.698
C03222=1048.693,134.265,-87.779,170.897,35.623,156.698
C03223=1048.687,134.016,-87.759,170.896,35.621,156.697
C03224=1048.681,133.767,-87.737,170.893,35.619,156.697
C03225=1048.675,133.518,-87.715,170.891,35.617,156.697
C03226=1048.669,133.269,-87.695,170.889,35.616,156.696
C03227=1048.663,133.020,-87.674,170.888,35.614,156.696
C03228=1048.658,132.771,-87.653,170.886,35.612,156.696
C03229=1048.651,132.522,-87.632,170.884,35.610,156.695
C03230=1048.645,132.273,-87.611,170.881,35.608,156.695
C03231=1048.639,132.024,-87.590,170.880,35.606,156.695
C03232=1048.632,131.775,-87.569,170.878,35.604,156.694
C03233=1048.627,131.526,-87.548,170.876,35.602,156.694
C03234=1048.621,131.276,-87.527,170.874,35.601,156.694
C03235=1048.615,131.028,-87.507,170.872,35.599,156.693
C03236=1048.608,130.779,-87.486,170.871,35.597,156.693
C03237=1048.602,130.529,-87.465,170.868,35.595,156.693
C03238=1048.596,130.281,-87.444,170.866,35.594,156.692
C03239=1048.590,130.031,-87.423,170.864,35.592,156.692
C03240=1048.584,129.783,-87.403,170.863,35.590,156.692
C03241=1048.577,129.533,-87.382,170.861,35.588,156.691
C03242=1048.571,129.284,-87.361,170.859,35.586,156.691
C03243=1048.565,129.035,-87.341,170.856,35.584,156.691
C03244=1048.559,128.786,-87.320,170.855,35.582,156.690
C03245=1048.553,128.537,-87.299,170.853,35.581,156.690
C03246=1048.546,128.288,-87.279,170.851,35.579,156.690
C03247=1048.541,128.039,-87.257,170.849,35.577,156.689
C03248=1048.534,127.789,-87.237,170.848,35.575,156.689
C03249=1048.528,127.541,-87.217,170.846,35.573,156.689
C03250=1048.522,127.291,-87.196,170.843,35.572,156.688
C03251=1048.516,127.043,-87.176,170.841,35.570,156.688
C03252=1048.509,126.794,-87.155,170.840,35.568,156.688
C03253=1048.503,126.544,-87.134,170.838,35.567,156.687
C03254=1048.497,126.295,-87.114,170.836,35.565,156.687
C03255=1048.490,126.010,-87.090,170.834,35.562,156.687
C03256=1048.483,125.724,-87.066,170.832,35.560,156.686
C03257=1048.476,125.438,-87.042,170.829,35.558,156.686
C03258=1048.469,125.152,-87.019,170.827,35.556,156.685
C03259=1048.463,124.904,-86.998,170.825,35.554,156.685
C03260=1048.457,124.654,-86.978,170.824,35.553,156.685
C03261=1048.451,124.405,-86.958,170.822,35.551,156.685
C03262=1048.445,124.156,-86.937,170.820,35.549,156.684
C03263=1048.439,123.907,-86.916,170.818,35.547,156.684
C03264=1048.432,123.658,-86.896,170.816,35.545,156.683
C03265=1048.427,123.409,-86.875,170.814,35.543,156.683
C03266=1048.420,123.159,-86.855,170.812,35.541,156.683
C03267=1048.414,122.911,-86.834,170.811,35.539,156.682
C03268=1048.408,122.661,-86.813,170.809,35.538,156.682
C03269=1048.402,122.412,-86.793,170.807,35.536,156.682
C03270=1048.396,122.164,-86.774,170.805,35.534,156.682
C03271=1048.389,121.915,-86.752,170.803,35.533,156.681
C03272=1048.384,121.666,-86.732,170.801,35.531,156.681
C03273=1048.377,121.416,-86.712,170.799,35.529,156.680
C03274=1048.371,121.167,-86.692,170.798,35.527,156.680
C03275=1048.365,120.917,-86.671,170.796,35.525,156.680
C03276=1048.359,120.669,-86.651,170.794,35.523,156.679
C03277=1048.353,120.420,-86.630,170.792,35.521,156.679
C03278=1048.347,120.171,-86.609,170.790,35.519,156.679
C03279=1048.341,119.922,-86.589,170.788,35.517,156.678
C03280=1048.335,119.673,-86.569,170.786,35.515,156.678
C03281=1048.329,119.423,-86.548,170.785,35.514,156.678
C03282=1048.323,119.174,-86.528,170.783,35.512,156.677
C03283=1048.317,118.925,-86.508,170.781,35.510,156.677
C03284=1048.311,118.676,-86.488,170.779,35.509,156.677
C03285=1048.305,118.427,-86.467,170.777,35.507,156.676
C03286=1048.299,118.178,-86.447,170.775,35.505,156.676
C03287=1048.293,117.929,-86.427,170.774,35.503,156.676
C03288=1048.287,117.680,-86.406,170.772,35.501,156.675
C03289=1048.281,117.431,-86.386,170.770,35.499,156.675
C03290=1048.275,117.182,-86.366,170.768,35.497,156.675
C03291=1048.269,116.933,-86.346,170.766,35.495,156.674
C03292=1048.263,116.683,-86.325,170.764,35.493,156.674
C03293=1048.257,116.434,-86.305,170.763,35.492,156.674
C03294=1048.251,116.185,-86.285,170.761,35.490,156.673
C03295=1048.245,115.936,-86.264,170.759,35.488,156.673
C03296=1048.239,115.687,-86.244,170.758,35.486,156.673
C03297=1048.233,115.438,-86.224,170.755,35.484,156.672
C03298=1048.227,115.189,-86.204,170.753,35.482,156.672
C03299=1048.221,114.939,-86.183,170.752,35.480,156.672
C03300=1048.215,114.691,-86.163,170.750,35.479,156.671
C03301=1048.209,114.442,-86.143,170.748,35.477,156.671
C03302=1048.203,114.192,-86.123,170.747,35.475,156.671
C03303=1048.198,113.943,-86.102,170.745,35.473,156.670
C03304=1048.192,113.694,-86.082,170.742,35.471,156.670
C03305=1048.185,113.445,-86.062,170.740,35.469,156.670
C03306=1048.179,113.195,-86.043,170.739,35.468,156.669
C03307=1048.173,112.947,-86.023,170.737,35.466,156.669
C03308=1048.167,112.698,-86.003,170.735,35.464,156.669
C03309=1048.161,112.448,-85.983,170.734,35.462,156.668
C03310=1048.155,112.199,-85.963,170.732,35.461,156.668
C03311=1048.149,111.951,-85.943,170.729,35.459,156.668
C03312=1048.142,111.700,-85.923,170.728,35.457,156.667
C03313=1048.136,111.452,-85.903,170.726,35.455,156.667
C03314=1048.130,111.203,-85.883,170.724,35.453,156.667
C03315=1048.124,110.953,-85.863,170.723,35.452,156.666
C03316=1048.118,110.704,-85.843,170.721,35.450,156.666
C03317=1048.112,110.455,-85.824,170.719,35.448,156.666
C03318=1048.106,110.206,-85.804,170.718,35.446,156.665
C03319=1048.099,109.921,-85.781,170.715,35.444,156.665
C03320=1048.092,109.634,-85.758,170.713,35.442,156.665
C03321=1048.085,109.349,-85.736,170.711,35.440,156.664
C03322=1048.078,109.063,-85.712,170.709,35.438,156.664
C03323=1048.071,108.813,-85.693,170.707,35.436,156.664
C03324=1048.065,108.565,-85.673,170.706,35.435,156.663
C03325=1048.059,108.316,-85.653,170.703,35.433,156.663
C03326=1048.052,108.066,-85.634,170.701,35.431,156.663
C03327=1048.046,107.817,-85.614,170.700,35.430,156.662
C03328=1048.040,107.568,-85.594,170.698,35.428,156.662
C03329=1048.035,107.319,-85.575,170.696,35.426,156.662
C03330=1048.028,107.069,-85.554,170.695,35.424,156.661
C03331=1048.021,106.821,-85.535,170.693,35.422,156.661
C03332=1048.016,106.571,-85.516,170.691,35.421,156.661
C03333=1048.010,106.322,-85.496,170.689,35.419,156.660
C03334=1048.004,106.074,-85.476,170.687,35.417,156.660
C03335=1047.997,105.824,-85.456,170.685,35.415,156.660
C03336=1047.991,105.575,-85.436,170.684,35.413,156.659
C03337=1047.985,105.326,-85.418,170.682,35.412,156.659
C03338=1047.979,105.077,-85.398,170.680,35.410,156.659
C03339=1047.973,104.828,-85.378,170.679,35.408,156.659
C03340=1047.967,104.578,-85.358,170.676,35.406,156.658
C03341=1047.961,104.329,-85.338,170.674,35.404,156.658
C03342=1047.955,104.080,-85.319,170.673,35.403,156.658
C03343=1047.948,103.831,-85.300,170.671,35.401,156.657
C03344=1047.942,103.582,-85.280,170.669,35.399,156.657
C03345=1047.936,103.332,-85.260,170.668,35.397,156.657
C03346=1047.930,103.083,-85.241,170.666,35.395,156.656
C03347=1047.924,102.834,-85.221,170.664,35.394,156.656
C03348=1047.918,102.585,-85.202,170.662,35.392,156.656
C03349=1047.912,102.336,-85.182,170.660,35.390,156.655
C03350=1047.906,102.087,-85.163,170.658,35.388,156.655
C03351=1047.900,101.838,-85.143,170.657,35.386,156.655
C03352=1047.894,101.588,-85.123,170.655,35.385,156.654
C03353=1047.888,101.339,-85.103,170.653,35.383,156.654
C03354=1047.881,101.090,-85.085,170.652,35.381,156.654
C03355=1047.875,100.841,-85.065,170.650,35.379,156.653
C03356=1047.870,100.591,-85.046,170.648,35.378,156.653
C03357=1047.863,100.343,-85.026,170.646,35.376,156.653
C03358=1047.857,100.093,-85.007,170.644,35.374,156.652
C03359=1047.851,99.843,-84.987,170.643,35.372,156.652
C03360=1047.844,99.595,-84.968,170.641,35.371,156.652
C03361=1047.839,99.345,-84.949,170.639,35.369,156.652
C03362=1047.832,99.097,-84.929,170.638,35.367,156.651
C03363=1047.826,98.847,-84.910,170.635,35.365,156.651
C03364=1047.820,98.598,-84.891,170.633,35.364,156.651
C03365=1047.814,98.350,-84.872,170.632,35.362,156.650
C03366=1047.807,98.099,-84.852,170.630,35.360,156.650
C03367=1047.801,97.850,-84.833,170.628,35.358,156.650
C03368=1047.795,97.601,-84.813,170.627,35.357,156.649
C03369=1047.789,97.352,-84.795,170.625,35.355,156.649
C03370=1047.783,97.103,-84.775,170.623,35.353,156.649
C03371=1047.776,96.854,-84.756,170.622,35.352,156.649
C03372=1047.770,96.605,-84.737,170.619,35.350,156.648
C03373=1047.764,96.356,-84.718,170.617,35.348,156.648
C03374=1047.758,96.106,-84.699,170.616,35.346,156.647
C03375=1047.752,95.857,-84.679,170.614,35.345,156.647
C03376=1047.745,95.608,-84.660,170.612,35.343,156.647
C03377=1047.740,95.358,-84.641,170.611,35.341,156.647
C03378=1047.733,95.109,-84.622,170.609,35.339,156.646
C03379=1047.727,94.860,-84.602,170.607,35.338,156.646
C03380=1047.721,94.611,-84.583,170.605,35.336,156.646
C03381=1047.715,94.362,-84.564,170.603,35.334,156.645
C03382=1047.709,94.113,-84.546,170.602,35.333,156.645
C03383=1047.701,93.827,-84.523,170.600,35.330,156.645
C03384=1047.695,93.541,-84.502,170.598,35.328,156.644
C03385=1047.688,93.255,-84.479,170.596,35.327,156.644
C03386=1047.681,92.969,-84.457,170.594,35.325,156.644
C03387=1047.674,92.720,-84.439,170.591,35.323,156.643
C03388=1047.668,92.471,-84.419,170.590,35.321,156.643
C03389=1047.662,92.222,-84.400,170.588,35.320,156.643
C03390=1047.656,91.973,-84.381,170.587,35.318,156.642
C03391=1047.650,91.723,-84.362,170.585,35.316,156.642
C03392=1047.644,91.474,-84.343,170.583,35.314,156.642
C03393=1047.638,91.225,-84.324,170.582,35.313,156.641
C03394=1047.632,90.975,-84.305,170.580,35.311,156.641
C03395=1047.625,90.727,-84.286,170.577,35.309,156.641
C03396=1047.620,90.478,-84.266,170.576,35.307,156.640
C03397=1047.613,90.228,-84.248,170.574,35.306,156.640
C03398=1047.607,89.979,-84.229,170.573,35.304,156.640
C03399=1047.601,89.730,-84.210,170.571,35.302,156.640
C03400=1047.595,89.481,-84.191,170.569,35.300,156.639
C03401=1047.588,89.232,-84.173,170.568,35.299,156.639
C03402=1047.583,88.982,-84.153,170.566,35.297,156.639
C03403=1047.576,88.733,-84.135,170.563,35.295,156.638
C03404=1047.570,88.484,-84.116,170.562,35.293,156.638
C03405=1047.563,88.235,-84.097,170.560,35.292,156.638
C03406=1047.558,87.985,-84.078,170.558,35.290,156.638
C03407=1047.551,87.736,-84.060,170.557,35.288,156.637
C03408=1047.545,87.487,-84.041,170.555,35.287,156.637
C03409=1047.538,87.238,-84.022,170.553,35.285,156.637
C03410=1047.533,86.989,-84.003,170.552,35.283,156.636
C03411=1047.526,86.739,-83.984,170.550,35.282,156.636
C03412=1047.520,86.490,-83.966,170.547,35.280,156.636
C03413=1047.514,86.241,-83.948,170.546,35.278,156.635
C03414=1047.507,85.991,-83.929,170.544,35.277,156.635
C03415=1047.502,85.742,-83.910,170.543,35.275,156.635
C03416=1047.495,85.493,-83.891,170.541,35.274,156.635
C03417=1047.489,85.244,-83.873,170.539,35.272,156.634
C03418=1047.482,84.995,-83.854,170.538,35.270,156.634
C03419=1047.477,84.745,-83.835,170.536,35.268,156.634
C03420=1047.470,84.496,-83.816,170.533,35.267,156.633
C03421=1047.464,84.247,-83.797,170.532,35.265,156.633
C03422=1047.458,83.998,-83.780,170.530,35.263,156.633
C03423=1047.453,83.749,-83.761,170.529,35.261,156.632
C03424=1047.446,83.499,-83.742,170.527,35.260,156.632
C03425=1047.440,83.250,-83.723,170.525,35.258,156.632
C03426=1047.433,83.001,-83.705,170.524,35.256,156.632
C03427=1047.427,82.752,-83.686,170.522,35.254,156.631
C03428=1047.422,82.502,-83.667,170.520,35.253,156.631
C03429=1047.415,82.253,-83.649,170.518,35.251,156.631
C03430=1047.409,82.004,-83.630,170.516,35.249,156.630
C03431=1047.402,81.755,-83.612,170.514,35.247,156.630
C03432=1047.396,81.506,-83.593,170.513,35.246,156.630
C03433=1047.391,81.256,-83.575,170.511,35.244,156.629
C03434=1047.385,81.007,-83.556,170.510,35.242,156.629
C03435=1047.378,80.758,-83.537,170.508,35.241,156.629
C03436=1047.372,80.509,-83.519,170.506,35.239,156.628
C03437=1047.366,80.259,-83.501,170.504,35.237,156.628
C03438=1047.360,80.010,-83.482,170.502,35.236,156.628
C03439=1047.354,79.761,-83.463,170.501,35.234,156.628
C03440=1047.348,79.512,-83.445,170.499,35.232,156.627
C03441=1047.342,79.262,-83.427,170.497,35.231,156.627
C03442=1047.335,79.013,-83.408,170.496,35.229,156.627
C03443=1047.329,78.764,-83.389,170.494,35.227,156.626
C03444=1047.323,78.514,-83.371,170.492,35.225,156.626
C03445=1047.317,78.265,-83.352,170.491,35.224,156.626
C03446=1047.311,78.017,-83.334,170.488,35.222,156.625
C03447=1047.303,77.730,-83.313,170.486,35.220,156.625
C03448=1047.297,77.444,-83.292,170.484,35.218,156.625
C03449=1047.289,77.158,-83.271,170.483,35.216,156.624
C03450=1047.283,76.873,-83.250,170.481,35.214,156.624
C03451=1047.276,76.623,-83.231,170.479,35.213,156.624
C03452=1047.270,76.374,-83.214,170.477,35.211,156.624
C03453=1047.264,76.125,-83.195,170.476,35.209,156.623
C03454=1047.257,75.876,-83.176,170.473,35.208,156.623
C03455=1047.252,75.626,-83.159,170.471,35.206,156.623
C03456=1047.245,75.377,-83.140,170.470,35.204,156.622
C03457=1047.238,75.128,-83.123,170.468,35.202,156.622
C03458=1047.232,74.879,-83.104,170.467,35.201,156.622
C03459=1047.226,74.629,-83.086,170.465,35.199,156.622
C03460=1047.220,74.381,-83.068,170.463,35.197,156.621
C03461=1047.214,74.131,-83.050,170.462,35.196,156.621
C03462=1047.207,73.882,-83.031,170.460,35.194,156.621
C03463=1047.201,73.632,-83.013,170.457,35.192,156.620
C03464=1047.195,73.383,-82.995,170.456,35.191,156.620
C03465=1047.189,73.134,-82.977,170.454,35.189,156.620
C03466=1047.183,72.885,-82.958,170.453,35.188,156.619
C03467=1047.177,72.635,-82.940,170.451,35.186,156.619
C03468=1047.170,72.386,-82.922,170.449,35.184,156.619
C03469=1047.165,72.137,-82.904,170.448,35.183,156.619
C03470=1047.158,71.888,-82.886,170.446,35.181,156.618
C03471=1047.152,71.638,-82.868,170.444,35.179,156.618
C03472=1047.145,71.389,-82.850,170.443,35.177,156.618
C03473=1047.139,71.139,-82.832,170.440,35.176,156.617
C03474=1047.134,70.890,-82.814,170.439,35.174,156.617
C03475=1047.127,70.641,-82.795,170.437,35.172,156.617
C03476=1047.121,70.392,-82.778,170.435,35.171,156.617
C03477=1047.115,70.142,-82.759,170.434,35.169,156.616
C03478=1047.109,69.893,-82.741,170.432,35.167,156.616
C03479=1047.102,69.644,-82.724,170.430,35.166,156.616
C03480=1047.096,69.395,-82.705,170.429,35.164,156.615
C03481=1047.090,69.146,-82.688,170.427,35.163,156.615
C03482=1047.084,68.896,-82.670,170.424,35.161,156.615
C03483=1047.078,68.647,-82.651,170.423,35.159,156.614
C03484=1047.071,68.397,-82.634,170.421,35.157,156.614
C03485=1047.065,68.148,-82.616,170.420,35.156,156.614
C03486=1047.059,67.899,-82.598,170.418,35.154,156.614
C03487=1047.053,67.650,-82.580,170.416,35.152,156.613
C03488=1047.046,67.400,-82.562,170.415,35.151,156.613
C03489=1047.040,67.152,-82.544,170.413,35.149,156.613
C03490=1047.034,66.902,-82.526,170.411,35.148,156.613
C03491=1047.028,66.652,-82.508,170.409,35.146,156.612
C03492=1047.022,66.404,-82.491,170.407,35.144,156.612
C03493=1047.015,66.154,-82.473,170.405,35.143,156.612
C03494=1047.009,65.905,-82.455,170.404,35.141,156.611
C03495=1047.003,65.656,-82.438,170.402,35.139,156.611
C03496=1046.997,65.406,-82.420,170.401,35.138,156.611
C03497=1046.990,65.157,-82.401,170.399,35.136,156.611
C03498=1046.983,64.908,-82.384,170.397,35.134,156.610
C03499=1046.978,64.659,-82.366,170.396,35.133,156.610
C03500=1046.972,64.409,-82.348,170.394,35.131,156.610
C03501=1046.966,64.159,-82.330,170.391,35.129,156.609
C03502=1046.959,63.910,-82.313,170.390,35.128,156.609
C03503=1046.953,63.661,-82.295,170.388,35.127,156.609
C03504=1046.946,63.412,-82.277,170.386,35.125,156.609
C03505=1046.939,63.162,-82.260,170.385,35.123,156.608
C03506=1046.934,62.913,-82.242,170.383,35.121,156.608
C03507=1046.927,62.664,-82.225,170.381,35.120,156.608
C03508=1046.921,62.414,-82.207,170.380,35.118,156.607
C03509=1046.915,62.165,-82.190,170.378,35.117,156.607
C03510=1046.908,61.916,-82.172,170.376,35.116,156.607
C03511=1046.901,61.630,-82.152,170.374,35.114,156.607
C03512=1046.893,61.344,-82.132,170.372,35.112,156.606
C03513=1046.886,61.058,-82.112,170.370,35.110,156.606
C03514=1046.879,60.772,-82.092,170.368,35.108,156.606
C03515=1046.873,60.522,-82.074,170.366,35.106,156.605
C03516=1046.866,60.273,-82.057,170.365,35.105,156.605
C03517=1046.860,60.024,-82.040,170.363,35.103,156.605
C03518=1046.854,59.775,-82.022,170.361,35.102,156.605
C03519=1046.847,59.525,-82.005,170.360,35.100,156.604
C03520=1046.841,59.276,-81.987,170.358,35.099,156.604
C03521=1046.834,59.027,-81.970,170.355,35.097,156.604
C03522=1046.828,58.777,-81.952,170.354,35.095,156.604
C03523=1046.822,58.528,-81.935,170.352,35.094,156.603
C03524=1046.815,58.279,-81.917,170.350,35.092,156.603
C03525=1046.810,58.030,-81.900,170.349,35.091,156.603
C03526=1046.803,57.780,-81.882,170.347,35.089,156.602
C03527=1046.797,57.531,-81.865,170.345,35.088,156.602
C03528=1046.790,57.282,-81.848,170.344,35.086,156.602
C03529=1046.783,57.032,-81.830,170.342,35.084,156.602
C03530=1046.778,56.783,-81.813,170.340,35.082,156.601
C03531=1046.771,56.533,-81.796,170.338,35.081,156.601
C03532=1046.765,56.284,-81.778,170.336,35.079,156.601
C03533=1046.759,56.035,-81.761,170.334,35.078,156.601
C03534=1046.752,55.785,-81.744,170.333,35.077,156.600
C03535=1046.747,55.536,-81.726,170.331,35.075,156.600
C03536=1046.740,55.287,-81.709,170.329,35.073,156.600
C03537=1046.734,55.037,-81.691,170.328,35.071,156.599
C03538=1046.727,54.788,-81.674,170.326,35.070,156.599
C03539=1046.721,54.538,-81.657,170.324,35.068,156.599
C03540=1046.715,54.289,-81.640,170.323,35.067,156.599
C03541=1046.708,54.040,-81.622,170.321,35.065,156.598
C03542=1046.702,53.791,-81.605,170.318,35.064,156.598
C03543=1046.696,53.541,-81.588,170.317,35.062,156.598
C03544=1046.690,53.293,-81.571,170.315,35.060,156.598
C03545=1046.684,53.042,-81.553,170.314,35.059,156.597
C03546=1046.678,52.794,-81.536,170.312,35.057,156.597
C03547=1046.671,52.544,-81.519,170.310,35.055,156.597
C03548=1046.665,52.295,-81.501,170.309,35.054,156.597
C03549=1046.659,52.046,-81.484,170.307,35.052,156.596
C03550=1046.653,51.796,-81.468,170.305,35.051,156.596
C03551=1046.646,51.547,-81.450,170.304,35.049,156.596
C03552=1046.640,51.298,-81.433,170.301,35.047,156.595
C03553=1046.634,51.048,-81.415,170.299,35.046,156.595
C03554=1046.628,50.799,-81.399,170.298,35.044,156.595
C03555=1046.621,50.549,-81.381,170.296,35.042,156.595
C03556=1046.616,50.300,-81.364,170.294,35.041,156.594
C03557=1046.609,50.051,-81.347,170.293,35.039,156.594
C03558=1046.603,49.802,-81.330,170.291,35.038,156.594
C03559=1046.597,49.552,-81.312,170.289,35.036,156.593
C03560=1046.591,49.303,-81.295,170.288,35.035,156.593
C03561=1046.585,49.054,-81.279,170.286,35.033,156.593
C03562=1046.578,48.804,-81.261,170.284,35.031,156.593
C03563=1046.572,48.555,-81.244,170.282,35.029,156.592
C03564=1046.566,48.305,-81.228,170.280,35.028,156.592
C03565=1046.560,48.056,-81.210,170.279,35.026,156.592
C03566=1046.553,47.807,-81.193,170.277,35.025,156.592
C03567=1046.547,47.557,-81.176,170.275,35.023,156.591
C03568=1046.542,47.308,-81.159,170.274,35.022,156.591
C03569=1046.535,47.059,-81.142,170.272,35.020,156.591
C03570=1046.529,46.810,-81.125,170.270,35.018,156.590
C03571=1046.523,46.560,-81.107,170.269,35.016,156.590
C03572=1046.517,46.311,-81.090,170.267,35.015,156.590
C03573=1046.511,46.062,-81.074,170.264,35.013,156.590
C03574=1046.505,45.812,-81.056,170.263,35.012,156.589
C03575=1046.497,45.526,-81.038,170.261,35.010,156.589
C03576=1046.490,45.240,-81.018,170.259,35.008,156.589
C03577=1046.484,44.953,-80.998,170.257,35.006,156.588
C03578=1046.476,44.666,-80.979,170.255,35.004,156.588
C03579=1046.470,44.417,-80.962,170.253,35.003,156.588
C03580=1046.465,44.168,-80.944,170.252,35.001,156.587
C03581=1046.458,43.918,-80.928,170.250,34.999,156.587
C03582=1046.452,43.670,-80.911,170.248,34.997,156.587
C03583=1046.446,43.420,-80.894,170.246,34.996,156.587
C03584=1046.440,43.170,-80.876,170.244,34.994,156.586
C03585=1046.434,42.921,-80.860,170.242,34.993,156.586
C03586=1046.427,42.672,-80.843,170.241,34.991,156.586
C03587=1046.421,42.422,-80.827,170.239,34.990,156.586
C03588=1046.415,42.173,-80.810,170.237,34.988,156.585
C03589=1046.408,41.924,-80.793,170.236,34.986,156.585
C03590=1046.402,41.674,-80.777,170.234,34.985,156.585
C03591=1046.396,41.425,-80.760,170.232,34.983,156.585
C03592=1046.389,41.175,-80.743,170.231,34.982,156.584
C03593=1046.383,40.927,-80.726,170.229,34.981,156.584
C03594=1046.377,40.677,-80.710,170.227,34.979,156.584
C03595=1046.371,40.427,-80.693,170.225,34.977,156.584
C03596=1046.364,40.179,-80.676,170.223,34.975,156.583
C03597=1046.358,39.928,-80.660,170.221,34.974,156.583
C03598=1046.351,39.680,-80.643,170.220,34.973,156.583
C03599=1046.346,39.430,-80.626,170.218,34.971,156.582
C03600=1046.340,39.181,-80.610,170.216,34.969,156.582
C03601=1046.333,38.931,-80.592,170.215,34.967,156.582
C03602=1046.328,38.682,-80.576,170.213,34.966,156.582
C03603=1046.322,38.433,-80.560,170.211,34.965,156.581
C03604=1046.315,38.183,-80.542,170.210,34.963,156.581
C03605=1046.309,37.934,-80.526,170.208,34.962,156.581
C03606=1046.303,37.684,-80.510,170.205,34.960,156.581
C03607=1046.296,37.435,-80.493,170.204,34.958,156.580
C03608=1046.290,37.186,-80.476,170.202,34.957,156.580
C03609=1046.283,36.937,-80.461,170.200,34.955,156.580
C03610=1046.277,36.687,-80.444,170.198,34.954,156.580
C03611=1046.270,36.438,-80.427,170.197,34.952,156.579
C03612=1046.265,36.189,-80.411,170.195,34.950,156.579
